LIN {X 0,Y 249.279,Z 155.051,A -85,B 0,C 180,E1 -18895.148,E2 -18895.148} C_VEL
LIN {X 0,Y 249.67,Z 155.011,A -85,B 0,C 180,E1 -18898.387,E2 -18898.387} C_VEL
LIN {X 0,Y 249.663,Z 155.008,A -85,B 0,C 180,E1 -18901.613,E2 -18901.613} C_VEL
LIN {X 0,Y 249.424,Z 155.041,A -85,B 0,C 180,E1 -18906.545,E2 -18906.545} C_VEL
LIN {X 0,Y 249.344,Z 155.042,A -85,B 0,C 180,E1 -18909.737,E2 -18909.737} C_VEL
LIN {X 0,Y 249.16,Z 155.074,A -85,B 0,C 180,E1 -18914.706,E2 -18914.706} C_VEL
LIN {X 0,Y 249.108,Z 155.073,A -85,B 0,C 180,E1 -18918.08,E2 -18918.08} C_VEL
LIN {X 0,Y 249.082,Z 155.075,A -85,B 0,C 180,E1 -18921.519,E2 -18921.519} C_VEL
LIN {X 0,Y 249.086,Z 155.051,A -85,B 0,C 180,E1 -18925.46,E2 -18925.46} C_VEL
LIN {X 0,Y 249.038,Z 155.082,A -85,B 0,C 180,E1 -18928.974,E2 -18928.974} C_VEL
LIN {X 0,Y 249.028,Z 155.089,A -85,B 0,C 180,E1 -18932.426,E2 -18932.426} C_VEL
LIN {X 0,Y 249.046,Z 155.084,A -85,B 0,C 180,E1 -18936.343,E2 -18936.343} C_VEL
LIN {X 0,Y 249.026,Z 155.159,A -85,B 0,C 180,E1 -18939.615,E2 -18939.615} C_VEL
LIN {X 0,Y 249.925,Z 157.806,A -85,B 0,C 180,E1 -18939.982,E2 -18939.982} C_VEL
LIN {X 0,Y 252.085,Z 160.128,A -85,B 0,C 180,E1 -18940.669,E2 -18940.669} C_VEL
LIN {X 0,Y 252.72,Z 160.982,A -85,B 0,C 180,E1 -18940.874,E2 -18940.874} C_VEL
LIN {X 0,Y 254.881,Z 164.177,A -85,B 0,C 180,E1 -18941.57,E2 -18941.57} C_VEL
LIN {X 0,Y 256.285,Z 165.902,A -85,B 0,C 180,E1 -18941.996,E2 -18941.996} C_VEL
LIN {X 0,Y 264.754,Z 177.926,A -85,B 0,C 180,E1 -18944.469,E2 -18944.469} C_VEL
LIN {X 0,Y 273.524,Z 191.575,A -85,B 0,C 180,E1 -18946.809,E2 -18946.809} C_VEL
LIN {X 0,Y 280.062,Z 204.114,A -85,B 0,C 180,E1 -18948.485,E2 -18948.485} C_VEL
LIN {X 0,Y 285.989,Z 217.193,A -85,B 0,C 180,E1 -18949.959,E2 -18949.959} C_VEL
LIN {X 0,Y 281.284,Z 313.77,A -85,B 0,C 180,E1 -18952.312,E2 -18952.312} C_VEL
LIN {X 0,Y 279.771,Z 329.461,A -85,B 0,C 180,E1 -18952.923,E2 -18952.923} C_VEL
LIN {X 0,Y 277.923,Z 343.793,A -85,B 0,C 180,E1 -18953.765,E2 -18953.765} C_VEL
LIN {X 0,Y 275.593,Z 357.91,A -85,B 0,C 180,E1 -18954.874,E2 -18954.874} C_VEL
LIN {X 0,Y 272.986,Z 370.88,A -85,B 0,C 180,E1 -18956.17,E2 -18956.17} C_VEL
LIN {X 0,Y 269.885,Z 383.644,A -85,B 0,C 180,E1 -18957.735,E2 -18957.735} C_VEL
LIN {X 0,Y 266.362,Z 396.502,A -85,B 0,C 180,E1 -18959.694,E2 -18959.694} C_VEL
LIN {X 0,Y 262.829,Z 408.079,A -85,B 0,C 180,E1 -18961.868,E2 -18961.868} C_VEL
LIN {X 0,Y 259.552,Z 418.653,A -85,B 0,C 180,E1 -18964.327,E2 -18964.327} C_VEL
LIN {X 0,Y 256.387,Z 428.094,A -85,B 0,C 180,E1 -18967.007,E2 -18967.007} C_VEL
LIN {X 0,Y 253.645,Z 435.952,A -85,B 0,C 180,E1 -18969.736,E2 -18969.736} C_VEL
LIN {X 0,Y 251.289,Z 443.278,A -85,B 0,C 180,E1 -18972.923,E2 -18972.923} C_VEL
LIN {X 0,Y 249.398,Z 449.09,A -85,B 0,C 180,E1 -18976.141,E2 -18976.141} C_VEL
LIN {X 0,Y 248.473,Z 452.526,A -85,B 0,C 180,E1 -18978.58,E2 -18978.58} C_VEL
LIN {X 0,Y 247.639,Z 456.003,A -85,B 0,C 180,E1 -18981.842,E2 -18981.842} C_VEL
LIN {X 0,Y 247.133,Z 458.3,A -85,B 0,C 180,E1 -18985.106,E2 -18985.106} C_VEL
LIN {X 0,Y 246.994,Z 459.468,A -85,B 0,C 180,E1 -18988.37,E2 -18988.37} C_VEL
LIN {X 0,Y 246.994,Z 459.481,A -85,B 0,C 180,E1 -18991.631,E2 -18991.631} C_VEL
LIN {X 0,Y 247.133,Z 458.365,A -85,B 0,C 180,E1 -18994.894,E2 -18994.894} C_VEL
LIN {X 0,Y 247.628,Z 456.118,A -85,B 0,C 180,E1 -18998.158,E2 -18998.158} C_VEL
LIN {X 0,Y 248.446,Z 452.688,A -85,B 0,C 180,E1 -19001.421,E2 -19001.421} C_VEL
LIN {X 0,Y 249.796,Z 447.987,A -85,B 0,C 180,E1 -19004.668,E2 -19004.668} C_VEL
LIN {X 0,Y 251.742,Z 441.891,A -85,B 0,C 180,E1 -19007.884,E2 -19007.884} C_VEL
LIN {X 0,Y 254.321,Z 434.209,A -85,B 0,C 180,E1 -19011.054,E2 -19011.054} C_VEL
LIN {X 0,Y 257.162,Z 426.014,A -85,B 0,C 180,E1 -19013.773,E2 -19013.773} C_VEL
LIN {X 0,Y 260.532,Z 416.135,A -85,B 0,C 180,E1 -19016.43,E2 -19016.43} C_VEL
LIN {X 0,Y 263.613,Z 406.01,A -85,B 0,C 180,E1 -19018.678,E2 -19018.678} C_VEL
LIN {X 0,Y 266.589,Z 396.072,A -85,B 0,C 180,E1 -19020.496,E2 -19020.496} C_VEL
LIN {X 0,Y 270.04,Z 383.126,A -85,B 0,C 180,E1 -19022.465,E2 -19022.465} C_VEL
LIN {X 0,Y 273.18,Z 370.256,A -85,B 0,C 180,E1 -19024.025,E2 -19024.025} C_VEL
LIN {X 0,Y 275.934,Z 356.158,A -85,B 0,C 180,E1 -19025.409,E2 -19025.409} C_VEL
LIN {X 0,Y 278.343,Z 341.437,A -85,B 0,C 180,E1 -19026.509,E2 -19026.509} C_VEL
LIN {X 0,Y 280.226,Z 326.136,A -85,B 0,C 180,E1 -19027.345,E2 -19027.345} C_VEL
LIN {X 0,Y 281.517,Z 311.329,A -85,B 0,C 180,E1 -19027.878,E2 -19027.878} C_VEL
LIN {X 0,Y 285.259,Z 232.852,A -85,B 0,C 180,E1 -19029.796,E2 -19029.796} C_VEL
LIN {X 0,Y 286.027,Z 216.985,A -85,B 0,C 180,E1 -19030.178,E2 -19030.178} C_VEL
LIN {X 0,Y 278.236,Z 200.326,A -85,B 0,C 180,E1 -19032.122,E2 -19032.122} C_VEL
LIN {X 0,Y 272.973,Z 190.671,A -85,B 0,C 180,E1 -19033.478,E2 -19033.478} C_VEL
LIN {X 0,Y 264.56,Z 177.55,A -85,B 0,C 180,E1 -19035.742,E2 -19035.742} C_VEL
LIN {X 0,Y 258.212,Z 168.659,A -85,B 0,C 180,E1 -19037.575,E2 -19037.575} C_VEL
LIN {X 0,Y 255.212,Z 164.469,A -85,B 0,C 180,E1 -19038.496,E2 -19038.496} C_VEL
LIN {X 0,Y 253.025,Z 161.57,A -85,B 0,C 180,E1 -19039.186,E2 -19039.186} C_VEL
LIN {X 0,Y 252.124,Z 160.16,A -85,B 0,C 180,E1 -19039.486,E2 -19039.486} C_VEL
LIN {X 0,Y 250.043,Z 158.023,A -85,B 0,C 180,E1 -19040.145,E2 -19040.145} C_VEL
LIN {X 0,Y 249.052,Z 155.413,A -85,B 0,C 180,E1 -19040.537,E2 -19040.537} C_VEL
LIN {X 0,Y 248.992,Z 155.088,A -85,B 0,C 180,E1 -19040.574,E2 -19040.574} C_VEL
LIN {X 0,Y 249.044,Z 155.083,A -85,B 0,C 180,E1 -19044.923,E2 -19044.923} C_VEL
LIN {X 0,Y 249.032,Z 155.058,A -85,B 0,C 180,E1 -19047.848,E2 -19047.848} C_VEL
LIN {X 0,Y 249.037,Z 155.083,A -85,B 0,C 180,E1 -19051.331,E2 -19051.331} C_VEL
LIN {X 0,Y 249.058,Z 155.082,A -85,B 0,C 180,E1 -19054.958,E2 -19054.958} C_VEL
LIN {X 0,Y 248.998,Z 155.084,A -85,B 0,C 180,E1 -19057.604,E2 -19057.604} C_VEL
LIN {X 0,Y 248.358,Z 155.171,A -85,B 0,C 180,E1 -19058.954,E2 -19058.954} C_VEL
LIN {X 0,Y 245.535,Z 155.517,A -85,B 0,C 180,E1 -19061.157,E2 -19061.157} C_VEL
LIN {X 0,Y 243.154,Z 155.815,A -85,B 0,C 180,E1 -19062.951,E2 -19062.951} C_VEL
LIN {X 0,Y 242.174,Z 155.944,A -85,B 0,C 180,E1 -19064.342,E2 -19064.342} C_VEL
LIN {X 0,Y 242.118,Z 155.947,A -85,B 0,C 180,E1 -19064.812,E2 -19064.812} C_VEL
LIN {X 0,Y 242.344,Z 155.909,A -85,B 0,C 180,E1 -19070.404,E2 -19070.404} C_VEL
LIN {X 0,Y 242.398,Z 155.917,A -85,B 0,C 180,E1 -19073.34,E2 -19073.34} C_VEL
LIN {X 0,Y 242.622,Z 155.886,A -85,B 0,C 180,E1 -19078.34,E2 -19078.34} C_VEL
LIN {X 0,Y 242.632,Z 155.883,A -85,B 0,C 180,E1 -19081.66,E2 -19081.66} C_VEL
LIN {X 0,Y 242.405,Z 155.915,A -85,B 0,C 180,E1 -19086.659,E2 -19086.659} C_VEL
LIN {X 0,Y 242.269,Z 155.923,A -85,B 0,C 180,E1 -19090.023,E2 -19090.023} C_VEL
LIN {X 0,Y 242.141,Z 155.945,A -85,B 0,C 180,E1 -19095.142,E2 -19095.142} C_VEL
LIN {X 0,Y 242.059,Z 155.949,A -85,B 0,C 180,E1 -19098.625,E2 -19098.625} C_VEL
LIN {X 0,Y 242.006,Z 155.956,A -85,B 0,C 180,E1 -19102.18,E2 -19102.18} C_VEL
LIN {X 0,Y 242.034,Z 155.954,A -85,B 0,C 180,E1 -19105.821,E2 -19105.821} C_VEL
LIN {X 0,Y 241.972,Z 155.969,A -85,B 0,C 180,E1 -19109.588,E2 -19109.588} C_VEL
LIN {X 0,Y 241.98,Z 155.958,A -85,B 0,C 180,E1 -19113.492,E2 -19113.492} C_VEL
LIN {X 0,Y 242.015,Z 156.047,A -85,B 0,C 180,E1 -19115.736,E2 -19115.736} C_VEL
LIN {X 0,Y 243.277,Z 159.716,A -85,B 0,C 180,E1 -19117.625,E2 -19117.625} C_VEL
LIN {X 0,Y 246.451,Z 164.423,A -85,B 0,C 180,E1 -19118.781,E2 -19118.781} C_VEL
LIN {X 0,Y 251.53,Z 172.11,A -85,B 0,C 180,E1 -19120.521,E2 -19120.521} C_VEL
LIN {X 0,Y 257.815,Z 182.158,A -85,B 0,C 180,E1 -19122.525,E2 -19122.525} C_VEL
LIN {X 0,Y 265.356,Z 195.282,A -85,B 0,C 180,E1 -19124.756,E2 -19124.756} C_VEL
LIN {X 0,Y 273.059,Z 210.704,A -85,B 0,C 180,E1 -19126.899,E2 -19126.899} C_VEL
LIN {X 0,Y 279.533,Z 225.506,A -85,B 0,C 180,E1 -19128.619,E2 -19128.619} C_VEL
LIN {X 0,Y 280.218,Z 227.267,A -85,B 0,C 180,E1 -19128.8,E2 -19128.8} C_VEL
LIN {X 0,Y 275.438,Z 323.887,A -85,B 0,C 180,E1 -19131.19,E2 -19131.19} C_VEL
LIN {X 0,Y 273.972,Z 339.511,A -85,B 0,C 180,E1 -19131.767,E2 -19131.767} C_VEL
LIN {X 0,Y 271.831,Z 354.535,A -85,B 0,C 180,E1 -19132.585,E2 -19132.585} C_VEL
LIN {X 0,Y 269.274,Z 368.105,A -85,B 0,C 180,E1 -19133.575,E2 -19133.575} C_VEL
LIN {X 0,Y 266.389,Z 381.613,A -85,B 0,C 180,E1 -19134.871,E2 -19134.871} C_VEL
LIN {X 0,Y 262.91,Z 395.389,A -85,B 0,C 180,E1 -19136.541,E2 -19136.541} C_VEL
LIN {X 0,Y 259.39,Z 407.401,A -85,B 0,C 180,E1 -19138.335,E2 -19138.335} C_VEL
LIN {X 0,Y 255.896,Z 418.533,A -85,B 0,C 180,E1 -19140.372,E2 -19140.372} C_VEL
LIN {X 0,Y 252.486,Z 429.103,A -85,B 0,C 180,E1 -19142.749,E2 -19142.749} C_VEL
LIN {X 0,Y 249.285,Z 438.815,A -85,B 0,C 180,E1 -19145.427,E2 -19145.427} C_VEL
LIN {X 0,Y 246.303,Z 447.143,A -85,B 0,C 180,E1 -19148.226,E2 -19148.226} C_VEL
LIN {X 0,Y 243.715,Z 454.975,A -85,B 0,C 180,E1 -19151.506,E2 -19151.506} C_VEL
LIN {X 0,Y 241.836,Z 461.213,A -85,B 0,C 180,E1 -19154.838,E2 -19154.838} C_VEL
LIN {X 0,Y 240.569,Z 466.043,A -85,B 0,C 180,E1 -19158.2,E2 -19158.2} C_VEL
LIN {X 0,Y 239.938,Z 469.588,A -85,B 0,C 180,E1 -19161.578,E2 -19161.578} C_VEL
LIN {X 0,Y 239.734,Z 472.123,A -85,B 0,C 180,E1 -19165.367,E2 -19165.367} C_VEL
LIN {X 0,Y 239.828,Z 473.101,A -85,B 0,C 180,E1 -19168.321,E2 -19168.321} C_VEL
LIN {X 0,Y 239.89,Z 473.257,A -85,B 0,C 180,E1 -19170,E2 -19170} C_VEL
LIN {X 0,Y 239.743,Z 472.642,A -85,B 0,C 180,E1 -19173.361,E2 -19173.361} C_VEL
LIN {X 0,Y 239.785,Z 470.873,A -85,B 0,C 180,E1 -19176.733,E2 -19176.733} C_VEL
LIN {X 0,Y 240.221,Z 467.929,A -85,B 0,C 180,E1 -19180.11,E2 -19180.11} C_VEL
LIN {X 0,Y 241.154,Z 463.743,A -85,B 0,C 180,E1 -19183.482,E2 -19183.482} C_VEL
LIN {X 0,Y 242.591,Z 458.203,A -85,B 0,C 180,E1 -19186.84,E2 -19186.84} C_VEL
LIN {X 0,Y 244.884,Z 451.171,A -85,B 0,C 180,E1 -19190.145,E2 -19190.145} C_VEL
LIN {X 0,Y 247.87,Z 442.43,A -85,B 0,C 180,E1 -19193.388,E2 -19193.388} C_VEL
LIN {X 0,Y 250.802,Z 433.768,A -85,B 0,C 180,E1 -19196.004,E2 -19196.004} C_VEL
LIN {X 0,Y 254.136,Z 423.717,A -85,B 0,C 180,E1 -19198.492,E2 -19198.492} C_VEL
LIN {X 0,Y 258.072,Z 411.491,A -85,B 0,C 180,E1 -19200.932,E2 -19200.932} C_VEL
LIN {X 0,Y 261.822,Z 399.029,A -85,B 0,C 180,E1 -19202.927,E2 -19202.927} C_VEL
LIN {X 0,Y 265.257,Z 386.188,A -85,B 0,C 180,E1 -19204.586,E2 -19204.586} C_VEL
LIN {X 0,Y 268.498,Z 371.686,A -85,B 0,C 180,E1 -19206.082,E2 -19206.082} C_VEL
LIN {X 0,Y 271.35,Z 356.628,A -85,B 0,C 180,E1 -19207.259,E2 -19207.259} C_VEL
LIN {X 0,Y 273.622,Z 341.541,A -85,B 0,C 180,E1 -19208.115,E2 -19208.115} C_VEL
LIN {X 0,Y 275.223,Z 325.688,A -85,B 0,C 180,E1 -19208.728,E2 -19208.728} C_VEL
LIN {X 0,Y 280.137,Z 228.134,A -85,B 0,C 180,E1 -19211.137,E2 -19211.137} C_VEL
LIN {X 0,Y 279.833,Z 226.451,A -85,B 0,C 180,E1 -19211.247,E2 -19211.247} C_VEL
LIN {X 0,Y 273.593,Z 211.928,A -85,B 0,C 180,E1 -19212.9,E2 -19212.9} C_VEL
LIN {X 0,Y 266.604,Z 197.759,A -85,B 0,C 180,E1 -19214.824,E2 -19214.824} C_VEL
LIN {X 0,Y 259.313,Z 184.701,A -85,B 0,C 180,E1 -19216.95,E2 -19216.95} C_VEL
LIN {X 0,Y 253.146,Z 174.691,A -85,B 0,C 180,E1 -19218.873,E2 -19218.873} C_VEL
LIN {X 0,Y 249.875,Z 169.56,A -85,B 0,C 180,E1 -19219.956,E2 -19219.956} C_VEL
LIN {X 0,Y 246.144,Z 164.055,A -85,B 0,C 180,E1 -19221.242,E2 -19221.242} C_VEL
LIN {X 0,Y 243.202,Z 159.541,A -85,B 0,C 180,E1 -19222.319,E2 -19222.319} C_VEL
LIN {X 0,Y 242.005,Z 155.955,A -85,B 0,C 180,E1 -19224.263,E2 -19224.263} C_VEL
LIN {X 0,Y 241.977,Z 155.966,A -85,B 0,C 180,E1 -19228.48,E2 -19228.48} C_VEL
LIN {X 0,Y 242.01,Z 155.959,A -85,B 0,C 180,E1 -19232.313,E2 -19232.313} C_VEL
LIN {X 0,Y 242.059,Z 155.951,A -85,B 0,C 180,E1 -19236.016,E2 -19236.016} C_VEL
LIN {X 0,Y 242.039,Z 155.952,A -85,B 0,C 180,E1 -19239.608,E2 -19239.608} C_VEL
LIN {X 0,Y 242.165,Z 155.936,A -85,B 0,C 180,E1 -19243.278,E2 -19243.278} C_VEL
LIN {X 0,Y 242.152,Z 155.94,A -85,B 0,C 180,E1 -19246.574,E2 -19246.574} C_VEL
LIN {X 0,Y 242.343,Z 155.919,A -85,B 0,C 180,E1 -19250.405,E2 -19250.405} C_VEL
LIN {X 0,Y 242.4,Z 155.916,A -85,B 0,C 180,E1 -19253.34,E2 -19253.34} C_VEL
LIN {X 0,Y 242.631,Z 155.888,A -85,B 0,C 180,E1 -19258.34,E2 -19258.34} C_VEL
LIN {X 0,Y 242.623,Z 155.885,A -85,B 0,C 180,E1 -19261.66,E2 -19261.66} C_VEL
LIN {X 0,Y 242.399,Z 155.917,A -85,B 0,C 180,E1 -19266.66,E2 -19266.66} C_VEL
LIN {X 0,Y 242.267,Z 155.926,A -85,B 0,C 180,E1 -19270.024,E2 -19270.024} C_VEL
LIN {X 0,Y 242.114,Z 155.952,A -85,B 0,C 180,E1 -19275.144,E2 -19275.144} C_VEL
LIN {X 0,Y 242.047,Z 155.958,A -85,B 0,C 180,E1 -19278.626,E2 -19278.626} C_VEL
LIN {X 0,Y 242.005,Z 155.961,A -85,B 0,C 180,E1 -19282.181,E2 -19282.181} C_VEL
LIN {X 0,Y 242.034,Z 155.926,A -85,B 0,C 180,E1 -19285.821,E2 -19285.821} C_VEL
LIN {X 0,Y 241.97,Z 155.97,A -85,B 0,C 180,E1 -19289.588,E2 -19289.588} C_VEL
LIN {X 0,Y 241.98,Z 155.964,A -85,B 0,C 180,E1 -19293.493,E2 -19293.493} C_VEL
LIN {X 0,Y 241.995,Z 155.966,A -85,B 0,C 180,E1 -19297.581,E2 -19297.581} C_VEL
LIN {X 0,Y 242.867,Z 158.603,A -85,B 0,C 180,E1 -19297.974,E2 -19297.974} C_VEL
LIN {X 0,Y 244.856,Z 160.844,A -85,B 0,C 180,E1 -19298.675,E2 -19298.675} C_VEL
LIN {X 0,Y 245.688,Z 161.619,A -85,B 0,C 180,E1 -19298.954,E2 -19298.954} C_VEL
LIN {X 0,Y 247.867,Z 165.014,A -85,B 0,C 180,E1 -19299.73,E2 -19299.73} C_VEL
LIN {X 0,Y 249.467,Z 166.854,A -85,B 0,C 180,E1 -19300.254,E2 -19300.254} C_VEL
LIN {X 0,Y 252.09,Z 170.381,A -85,B 0,C 180,E1 -19301.109,E2 -19301.109} C_VEL
LIN {X 0,Y 261.02,Z 183.198,A -85,B 0,C 180,E1 -19303.827,E2 -19303.827} C_VEL
LIN {X 0,Y 269.645,Z 196.844,A -85,B 0,C 180,E1 -19306.216,E2 -19306.216} C_VEL
LIN {X 0,Y 276.191,Z 209.815,A -85,B 0,C 180,E1 -19307.961,E2 -19307.961} C_VEL
LIN {X 0,Y 280.5,Z 219.373,A -85,B 0,C 180,E1 -19309.075,E2 -19309.075} C_VEL
LIN {X 0,Y 275.708,Z 313.988,A -85,B 0,C 180,E1 -19311.411,E2 -19311.411} C_VEL
LIN {X 0,Y 274.139,Z 329.672,A -85,B 0,C 180,E1 -19312.028,E2 -19312.028} C_VEL
LIN {X 0,Y 272.063,Z 345.291,A -85,B 0,C 180,E1 -19312.971,E2 -19312.971} C_VEL
LIN {X 0,Y 269.525,Z 359.809,A -85,B 0,C 180,E1 -19314.159,E2 -19314.159} C_VEL
LIN {X 0,Y 266.398,Z 374.215,A -85,B 0,C 180,E1 -19315.674,E2 -19315.674} C_VEL
LIN {X 0,Y 262.879,Z 387.666,A -85,B 0,C 180,E1 -19317.45,E2 -19317.45} C_VEL
LIN {X 0,Y 259.283,Z 399.872,A -85,B 0,C 180,E1 -19319.454,E2 -19319.454} C_VEL
LIN {X 0,Y 255.626,Z 411.397,A -85,B 0,C 180,E1 -19321.798,E2 -19321.798} C_VEL
LIN {X 0,Y 252.133,Z 421.778,A -85,B 0,C 180,E1 -19324.402,E2 -19324.402} C_VEL
LIN {X 0,Y 249.01,Z 430.732,A -85,B 0,C 180,E1 -19327.165,E2 -19327.165} C_VEL
LIN {X 0,Y 246.233,Z 438.153,A -85,B 0,C 180,E1 -19329.97,E2 -19329.97} C_VEL
LIN {X 0,Y 243.968,Z 445.077,A -85,B 0,C 180,E1 -19333.258,E2 -19333.258} C_VEL
LIN {X 0,Y 242.116,Z 450.518,A -85,B 0,C 180,E1 -19336.572,E2 -19336.572} C_VEL
LIN {X 0,Y 240.984,Z 454.617,A -85,B 0,C 180,E1 -19339.922,E2 -19339.922} C_VEL
LIN {X 0,Y 240.273,Z 457.494,A -85,B 0,C 180,E1 -19343.281,E2 -19343.281} C_VEL
LIN {X 0,Y 239.977,Z 459.221,A -85,B 0,C 180,E1 -19346.642,E2 -19346.642} C_VEL
LIN {X 0,Y 239.922,Z 459.821,A -85,B 0,C 180,E1 -19350,E2 -19350} C_VEL
LIN {X 0,Y 239.977,Z 459.259,A -85,B 0,C 180,E1 -19353.358,E2 -19353.358} C_VEL
LIN {X 0,Y 240.273,Z 457.584,A -85,B 0,C 180,E1 -19356.719,E2 -19356.719} C_VEL
LIN {X 0,Y 240.943,Z 454.755,A -85,B 0,C 180,E1 -19360.079,E2 -19360.079} C_VEL
LIN {X 0,Y 242.07,Z 450.702,A -85,B 0,C 180,E1 -19363.43,E2 -19363.43} C_VEL
LIN {X 0,Y 243.928,Z 445.319,A -85,B 0,C 180,E1 -19366.745,E2 -19366.745} C_VEL
LIN {X 0,Y 246.216,Z 438.462,A -85,B 0,C 180,E1 -19370.031,E2 -19370.031} C_VEL
LIN {X 0,Y 249.294,Z 429.892,A -85,B 0,C 180,E1 -19373.246,E2 -19373.246} C_VEL
LIN {X 0,Y 252.548,Z 420.775,A -85,B 0,C 180,E1 -19375.995,E2 -19375.995} C_VEL
LIN {X 0,Y 255.556,Z 411.941,A -85,B 0,C 180,E1 -19378.194,E2 -19378.194} C_VEL
LIN {X 0,Y 259.144,Z 400.45,A -85,B 0,C 180,E1 -19380.564,E2 -19380.564} C_VEL
LIN {X 0,Y 262.729,Z 388.354,A -85,B 0,C 180,E1 -19382.571,E2 -19382.571} C_VEL
LIN {X 0,Y 265.927,Z 376.485,A -85,B 0,C 180,E1 -19384.167,E2 -19384.167} C_VEL
LIN {X 0,Y 268.756,Z 363.809,A -85,B 0,C 180,E1 -19385.578,E2 -19385.578} C_VEL
LIN {X 0,Y 271.362,Z 350.032,A -85,B 0,C 180,E1 -19386.792,E2 -19386.792} C_VEL
LIN {X 0,Y 273.568,Z 335.39,A -85,B 0,C 180,E1 -19387.774,E2 -19387.774} C_VEL
LIN {X 0,Y 275.265,Z 320.346,A -85,B 0,C 180,E1 -19388.487,E2 -19388.487} C_VEL
LIN {X 0,Y 276.424,Z 303.318,A -85,B 0,C 180,E1 -19388.996,E2 -19388.996} C_VEL
LIN {X 0,Y 280.525,Z 219.259,A -85,B 0,C 180,E1 -19391.063,E2 -19391.063} C_VEL
LIN {X 0,Y 272.917,Z 202.924,A -85,B 0,C 180,E1 -19393.054,E2 -19393.054} C_VEL
LIN {X 0,Y 267.7,Z 193.547,A -85,B 0,C 180,E1 -19394.458,E2 -19394.458} C_VEL
LIN {X 0,Y 259.333,Z 180.741,A -85,B 0,C 180,E1 -19396.82,E2 -19396.82} C_VEL
LIN {X 0,Y 254.1,Z 173.341,A -85,B 0,C 180,E1 -19398.409,E2 -19398.409} C_VEL
LIN {X 0,Y 251.807,Z 170.056,A -85,B 0,C 180,E1 -19399.145,E2 -19399.145} C_VEL
LIN {X 0,Y 249.225,Z 166.389,A -85,B 0,C 180,E1 -19400.002,E2 -19400.002} C_VEL
LIN {X 0,Y 246.478,Z 163.164,A -85,B 0,C 180,E1 -19400.92,E2 -19400.92} C_VEL
LIN {X 0,Y 245.414,Z 161.207,A -85,B 0,C 180,E1 -19401.319,E2 -19401.319} C_VEL
LIN {X 0,Y 243.17,Z 159.063,A -85,B 0,C 180,E1 -19402.09,E2 -19402.09} C_VEL
LIN {X 0,Y 242.146,Z 156.808,A -85,B 0,C 180,E1 -19402.512,E2 -19402.512} C_VEL
LIN {X 0,Y 241.958,Z 155.942,A -85,B 0,C 180,E1 -19402.642,E2 -19402.642} C_VEL
LIN {X 0,Y 241.98,Z 155.955,A -85,B 0,C 180,E1 -19406.507,E2 -19406.507} C_VEL
LIN {X 0,Y 241.972,Z 155.948,A -85,B 0,C 180,E1 -19410.615,E2 -19410.615} C_VEL
LIN {X 0,Y 241.997,Z 155.957,A -85,B 0,C 180,E1 -19414.197,E2 -19414.197} C_VEL
LIN {X 0,Y 241.987,Z 155.958,A -85,B 0,C 180,E1 -19418.338,E2 -19418.338} C_VEL
LIN {X 0,Y 242.115,Z 155.949,A -85,B 0,C 180,E1 -19423.318,E2 -19423.318} C_VEL
LIN {X 0,Y 242.118,Z 155.947,A -85,B 0,C 180,E1 -19424.812,E2 -19424.812} C_VEL
LIN {X 0,Y 241.526,Z 156.027,A -85,B 0,C 180,E1 -19426.202,E2 -19426.202} C_VEL
LIN {X 0,Y 238.758,Z 156.37,A -85,B 0,C 180,E1 -19428.472,E2 -19428.472} C_VEL
LIN {X 0,Y 236.381,Z 156.655,A -85,B 0,C 180,E1 -19430.321,E2 -19430.321} C_VEL
LIN {X 0,Y 235.376,Z 156.781,A -85,B 0,C 180,E1 -19431.754,E2 -19431.754} C_VEL
LIN {X 0,Y 235.304,Z 156.79,A -85,B 0,C 180,E1 -19432.24,E2 -19432.24} C_VEL
LIN {X 0,Y 235.581,Z 156.764,A -85,B 0,C 180,E1 -19438.29,E2 -19438.29} C_VEL
LIN {X 0,Y 235.591,Z 156.76,A -85,B 0,C 180,E1 -19441.709,E2 -19441.709} C_VEL
LIN {X 0,Y 235.357,Z 156.794,A -85,B 0,C 180,E1 -19446.86,E2 -19446.86} C_VEL
LIN {X 0,Y 235.216,Z 156.803,A -85,B 0,C 180,E1 -19450.327,E2 -19450.327} C_VEL
LIN {X 0,Y 235.088,Z 156.829,A -85,B 0,C 180,E1 -19455.608,E2 -19455.608} C_VEL
LIN {X 0,Y 234.999,Z 156.832,A -85,B 0,C 180,E1 -19459.206,E2 -19459.206} C_VEL
LIN {X 0,Y 234.951,Z 156.835,A -85,B 0,C 180,E1 -19462.884,E2 -19462.884} C_VEL
LIN {X 0,Y 234.948,Z 156.834,A -85,B 0,C 180,E1 -19466.66,E2 -19466.66} C_VEL
LIN {X 0,Y 234.901,Z 156.85,A -85,B 0,C 180,E1 -19470.572,E2 -19470.572} C_VEL
LIN {X 0,Y 234.953,Z 156.98,A -85,B 0,C 180,E1 -19473.896,E2 -19473.896} C_VEL
LIN {X 0,Y 235.708,Z 159.293,A -85,B 0,C 180,E1 -19475.163,E2 -19475.163} C_VEL
LIN {X 0,Y 239.209,Z 164.253,A -85,B 0,C 180,E1 -19476.574,E2 -19476.574} C_VEL
LIN {X 0,Y 244.827,Z 172.493,A -85,B 0,C 180,E1 -19478.679,E2 -19478.679} C_VEL
LIN {X 0,Y 248.268,Z 177.891,A -85,B 0,C 180,E1 -19479.893,E2 -19479.893} C_VEL
LIN {X 0,Y 254.035,Z 187.247,A -85,B 0,C 180,E1 -19481.804,E2 -19481.804} C_VEL
LIN {X 0,Y 261.151,Z 199.822,A -85,B 0,C 180,E1 -19484,E2 -19484} C_VEL
LIN {X 0,Y 268.925,Z 215.645,A -85,B 0,C 180,E1 -19486.253,E2 -19486.253} C_VEL
LIN {X 0,Y 274.781,Z 229.379,A -85,B 0,C 180,E1 -19487.878,E2 -19487.878} C_VEL
LIN {X 0,Y 270.599,Z 311.991,A -85,B 0,C 180,E1 -19489.937,E2 -19489.937} C_VEL
LIN {X 0,Y 269.322,Z 331.334,A -85,B 0,C 180,E1 -19490.5,E2 -19490.5} C_VEL
LIN {X 0,Y 267.41,Z 346.7,A -85,B 0,C 180,E1 -19491.196,E2 -19491.196} C_VEL
LIN {X 0,Y 264.858,Z 361.541,A -85,B 0,C 180,E1 -19492.148,E2 -19492.148} C_VEL
LIN {X 0,Y 261.969,Z 375.458,A -85,B 0,C 180,E1 -19493.351,E2 -19493.351} C_VEL
LIN {X 0,Y 258.562,Z 389.504,A -85,B 0,C 180,E1 -19494.92,E2 -19494.92} C_VEL
LIN {X 0,Y 254.73,Z 402.636,A -85,B 0,C 180,E1 -19496.746,E2 -19496.746} C_VEL
LIN {X 0,Y 250.993,Z 414.47,A -85,B 0,C 180,E1 -19498.801,E2 -19498.801} C_VEL
LIN {X 0,Y 247.311,Z 425.318,A -85,B 0,C 180,E1 -19501.112,E2 -19501.112} C_VEL
LIN {X 0,Y 243.652,Z 436.004,A -85,B 0,C 180,E1 -19503.941,E2 -19503.941} C_VEL
LIN {X 0,Y 240.458,Z 444.694,A -85,B 0,C 180,E1 -19506.76,E2 -19506.76} C_VEL
LIN {X 0,Y 238.16,Z 451.072,A -85,B 0,C 180,E1 -19509.261,E2 -19509.261} C_VEL
LIN {X 0,Y 235.824,Z 458.08,A -85,B 0,C 180,E1 -19512.661,E2 -19512.661} C_VEL
LIN {X 0,Y 234.202,Z 463.596,A -85,B 0,C 180,E1 -19516.109,E2 -19516.109} C_VEL
LIN {X 0,Y 233.167,Z 467.771,A -85,B 0,C 180,E1 -19519.581,E2 -19519.581} C_VEL
LIN {X 0,Y 232.705,Z 470.704,A -85,B 0,C 180,E1 -19523.061,E2 -19523.061} C_VEL
LIN {X 0,Y 232.651,Z 472.456,A -85,B 0,C 180,E1 -19526.536,E2 -19526.536} C_VEL
LIN {X 0,Y 232.801,Z 473.058,A -85,B 0,C 180,E1 -19530,E2 -19530} C_VEL
LIN {X 0,Y 232.651,Z 472.443,A -85,B 0,C 180,E1 -19533.464,E2 -19533.464} C_VEL
LIN {X 0,Y 232.705,Z 470.673,A -85,B 0,C 180,E1 -19536.939,E2 -19536.939} C_VEL
LIN {X 0,Y 233.166,Z 467.727,A -85,B 0,C 180,E1 -19540.419,E2 -19540.419} C_VEL
LIN {X 0,Y 234.189,Z 463.541,A -85,B 0,C 180,E1 -19543.891,E2 -19543.891} C_VEL
LIN {X 0,Y 235.804,Z 457.717,A -85,B 0,C 180,E1 -19547.496,E2 -19547.496} C_VEL
LIN {X 0,Y 238.155,Z 450.969,A -85,B 0,C 180,E1 -19550.74,E2 -19550.74} C_VEL
LIN {X 0,Y 240.836,Z 443.452,A -85,B 0,C 180,E1 -19553.656,E2 -19553.656} C_VEL
LIN {X 0,Y 243.906,Z 434.883,A -85,B 0,C 180,E1 -19556.362,E2 -19556.362} C_VEL
LIN {X 0,Y 247.304,Z 425.156,A -85,B 0,C 180,E1 -19558.889,E2 -19558.889} C_VEL
LIN {X 0,Y 250.965,Z 414.277,A -85,B 0,C 180,E1 -19561.203,E2 -19561.203} C_VEL
LIN {X 0,Y 254.725,Z 402.408,A -85,B 0,C 180,E1 -19563.255,E2 -19563.255} C_VEL
LIN {X 0,Y 258.549,Z 389.316,A -85,B 0,C 180,E1 -19565.065,E2 -19565.065} C_VEL
LIN {X 0,Y 261.569,Z 376.858,A -85,B 0,C 180,E1 -19566.475,E2 -19566.475} C_VEL
LIN {X 0,Y 264.43,Z 363.34,A -85,B 0,C 180,E1 -19567.683,E2 -19567.683} C_VEL
LIN {X 0,Y 267.076,Z 348.377,A -85,B 0,C 180,E1 -19568.68,E2 -19568.68} C_VEL
LIN {X 0,Y 268.965,Z 333.822,A -85,B 0,C 180,E1 -19569.38,E2 -19569.38} C_VEL
LIN {X 0,Y 270.196,Z 317.66,A -85,B 0,C 180,E1 -19569.891,E2 -19569.891} C_VEL
LIN {X 0,Y 274.664,Z 229.275,A -85,B 0,C 180,E1 -19572.095,E2 -19572.095} C_VEL
LIN {X 0,Y 268.778,Z 215.5,A -85,B 0,C 180,E1 -19573.725,E2 -19573.725} C_VEL
LIN {X 0,Y 262.197,Z 201.997,A -85,B 0,C 180,E1 -19575.619,E2 -19575.619} C_VEL
LIN {X 0,Y 255.557,Z 189.85,A -85,B 0,C 180,E1 -19577.642,E2 -19577.642} C_VEL
LIN {X 0,Y 249.108,Z 179.249,A -85,B 0,C 180,E1 -19579.741,E2 -19579.741} C_VEL
LIN {X 0,Y 246.409,Z 174.935,A -85,B 0,C 180,E1 -19580.675,E2 -19580.675} C_VEL
LIN {X 0,Y 242.638,Z 169.284,A -85,B 0,C 180,E1 -19582.031,E2 -19582.031} C_VEL
LIN {X 0,Y 239.165,Z 164.145,A -85,B 0,C 180,E1 -19583.352,E2 -19583.352} C_VEL
LIN {X 0,Y 235.967,Z 159.707,A -85,B 0,C 180,E1 -19584.628,E2 -19584.628} C_VEL
LIN {X 0,Y 235.483,Z 158.828,A -85,B 0,C 180,E1 -19584.936,E2 -19584.936} C_VEL
LIN {X 0,Y 234.93,Z 156.839,A -85,B 0,C 180,E1 -19586.203,E2 -19586.203} C_VEL
LIN {X 0,Y 234.971,Z 156.831,A -85,B 0,C 180,E1 -19590.157,E2 -19590.157} C_VEL
LIN {X 0,Y 234.995,Z 156.831,A -85,B 0,C 180,E1 -19593.794,E2 -19593.794} C_VEL
LIN {X 0,Y 235.013,Z 156.831,A -85,B 0,C 180,E1 -19598.97,E2 -19598.97} C_VEL
LIN {X 0,Y 235.098,Z 156.817,A -85,B 0,C 180,E1 -19603.06,E2 -19603.06} C_VEL
LIN {X 0,Y 235.106,Z 156.814,A -85,B 0,C 180,E1 -19607.922,E2 -19607.922} C_VEL
LIN {X 0,Y 235.313,Z 156.787,A -85,B 0,C 180,E1 -19611.412,E2 -19611.412} C_VEL
LIN {X 0,Y 235.351,Z 156.791,A -85,B 0,C 180,E1 -19613.14,E2 -19613.14} C_VEL
LIN {X 0,Y 235.591,Z 156.765,A -85,B 0,C 180,E1 -19618.291,E2 -19618.291} C_VEL
LIN {X 0,Y 235.581,Z 156.763,A -85,B 0,C 180,E1 -19621.71,E2 -19621.71} C_VEL
LIN {X 0,Y 235.35,Z 156.794,A -85,B 0,C 180,E1 -19626.86,E2 -19626.86} C_VEL
LIN {X 0,Y 235.213,Z 156.807,A -85,B 0,C 180,E1 -19630.328,E2 -19630.328} C_VEL
LIN {X 0,Y 235.066,Z 156.829,A -85,B 0,C 180,E1 -19635.61,E2 -19635.61} C_VEL
LIN {X 0,Y 234.989,Z 156.84,A -85,B 0,C 180,E1 -19639.207,E2 -19639.207} C_VEL
LIN {X 0,Y 234.947,Z 156.845,A -85,B 0,C 180,E1 -19642.884,E2 -19642.884} C_VEL
LIN {X 0,Y 234.946,Z 156.807,A -85,B 0,C 180,E1 -19646.66,E2 -19646.66} C_VEL
LIN {X 0,Y 234.9,Z 156.846,A -85,B 0,C 180,E1 -19650.573,E2 -19650.573} C_VEL
LIN {X 0,Y 234.93,Z 156.838,A -85,B 0,C 180,E1 -19654.638,E2 -19654.638} C_VEL
LIN {X 0,Y 234.941,Z 156.864,A -85,B 0,C 180,E1 -19655.313,E2 -19655.313} C_VEL
LIN {X 0,Y 235.76,Z 159.341,A -85,B 0,C 180,E1 -19655.722,E2 -19655.722} C_VEL
LIN {X 0,Y 237.753,Z 161.641,A -85,B 0,C 180,E1 -19656.505,E2 -19656.505} C_VEL
LIN {X 0,Y 238.842,Z 162.527,A -85,B 0,C 180,E1 -19656.903,E2 -19656.903} C_VEL
LIN {X 0,Y 240.78,Z 165.718,A -85,B 0,C 180,E1 -19657.672,E2 -19657.672} C_VEL
LIN {X 0,Y 242.623,Z 167.696,A -85,B 0,C 180,E1 -19658.329,E2 -19658.329} C_VEL
LIN {X 0,Y 245.298,Z 171.406,A -85,B 0,C 180,E1 -19659.288,E2 -19659.288} C_VEL
LIN {X 0,Y 252.299,Z 181.076,A -85,B 0,C 180,E1 -19661.617,E2 -19661.617} C_VEL
LIN {X 0,Y 260.424,Z 193.374,A -85,B 0,C 180,E1 -19664.087,E2 -19664.087} C_VEL
LIN {X 0,Y 266.474,Z 203.452,A -85,B 0,C 180,E1 -19665.798,E2 -19665.798} C_VEL
LIN {X 0,Y 273.417,Z 217.936,A -85,B 0,C 180,E1 -19667.715,E2 -19667.715} C_VEL
LIN {X 0,Y 275.057,Z 221.604,A -85,B 0,C 180,E1 -19668.154,E2 -19668.154} C_VEL
LIN {X 0,Y 270.201,Z 314.207,A -85,B 0,C 180,E1 -19670.473,E2 -19670.473} C_VEL
LIN {X 0,Y 268.578,Z 329.883,A -85,B 0,C 180,E1 -19671.096,E2 -19671.096} C_VEL
LIN {X 0,Y 266.435,Z 345.498,A -85,B 0,C 180,E1 -19672.053,E2 -19672.053} C_VEL
LIN {X 0,Y 264.044,Z 358.614,A -85,B 0,C 180,E1 -19673.126,E2 -19673.126} C_VEL
LIN {X 0,Y 260.945,Z 372.866,A -85,B 0,C 180,E1 -19674.616,E2 -19674.616} C_VEL
LIN {X 0,Y 257.284,Z 386.624,A -85,B 0,C 180,E1 -19676.416,E2 -19676.416} C_VEL
LIN {X 0,Y 253.521,Z 399.036,A -85,B 0,C 180,E1 -19678.45,E2 -19678.45} C_VEL
LIN {X 0,Y 249.703,Z 410.423,A -85,B 0,C 180,E1 -19680.752,E2 -19680.752} C_VEL
LIN {X 0,Y 246.826,Z 419.055,A -85,B 0,C 180,E1 -19682.898,E2 -19682.898} C_VEL
LIN {X 0,Y 243.328,Z 428.497,A -85,B 0,C 180,E1 -19685.696,E2 -19685.696} C_VEL
LIN {X 0,Y 240.334,Z 436.354,A -85,B 0,C 180,E1 -19688.56,E2 -19688.56} C_VEL
LIN {X 0,Y 238.224,Z 442.015,A -85,B 0,C 180,E1 -19691.064,E2 -19691.064} C_VEL
LIN {X 0,Y 236.085,Z 448.174,A -85,B 0,C 180,E1 -19694.459,E2 -19694.459} C_VEL
LIN {X 0,Y 234.527,Z 452.927,A -85,B 0,C 180,E1 -19697.891,E2 -19697.891} C_VEL
LIN {X 0,Y 233.558,Z 456.402,A -85,B 0,C 180,E1 -19701.347,E2 -19701.347} C_VEL
LIN {X 0,Y 232.989,Z 458.698,A -85,B 0,C 180,E1 -19704.808,E2 -19704.808} C_VEL
LIN {X 0,Y 232.821,Z 459.865,A -85,B 0,C 180,E1 -19708.27,E2 -19708.27} C_VEL
LIN {X 0,Y 232.821,Z 459.878,A -85,B 0,C 180,E1 -19711.73,E2 -19711.73} C_VEL
LIN {X 0,Y 233.03,Z 458.585,A -85,B 0,C 180,E1 -19715.581,E2 -19715.581} C_VEL
LIN {X 0,Y 233.526,Z 456.516,A -85,B 0,C 180,E1 -19718.655,E2 -19718.655} C_VEL
LIN {X 0,Y 234.471,Z 453.086,A -85,B 0,C 180,E1 -19722.112,E2 -19722.112} C_VEL
LIN {X 0,Y 236.058,Z 448.383,A -85,B 0,C 180,E1 -19725.543,E2 -19725.543} C_VEL
LIN {X 0,Y 238.185,Z 442.288,A -85,B 0,C 180,E1 -19728.94,E2 -19728.94} C_VEL
LIN {X 0,Y 241.054,Z 434.605,A -85,B 0,C 180,E1 -19732.273,E2 -19732.273} C_VEL
LIN {X 0,Y 244.171,Z 426.409,A -85,B 0,C 180,E1 -19735.122,E2 -19735.122} C_VEL
LIN {X 0,Y 247.856,Z 416.528,A -85,B 0,C 180,E1 -19737.896,E2 -19737.896} C_VEL
LIN {X 0,Y 251.188,Z 406.404,A -85,B 0,C 180,E1 -19740.24,E2 -19740.24} C_VEL
LIN {X 0,Y 254.768,Z 395.398,A -85,B 0,C 180,E1 -19742.309,E2 -19742.309} C_VEL
LIN {X 0,Y 258.176,Z 383.515,A -85,B 0,C 180,E1 -19744.156,E2 -19744.156} C_VEL
LIN {X 0,Y 261.528,Z 370.643,A -85,B 0,C 180,E1 -19745.767,E2 -19745.767} C_VEL
LIN {X 0,Y 264.531,Z 356.387,A -85,B 0,C 180,E1 -19747.203,E2 -19747.203} C_VEL
LIN {X 0,Y 267.062,Z 341.817,A -85,B 0,C 180,E1 -19748.322,E2 -19748.322} C_VEL
LIN {X 0,Y 269.105,Z 326.508,A -85,B 0,C 180,E1 -19749.175,E2 -19749.175} C_VEL
LIN {X 0,Y 270.458,Z 311.686,A -85,B 0,C 180,E1 -19749.724,E2 -19749.724} C_VEL
LIN {X 0,Y 274.52,Z 233.122,A -85,B 0,C 180,E1 -19751.693,E2 -19751.693} C_VEL
LIN {X 0,Y 275.093,Z 221.513,A -85,B 0,C 180,E1 -19751.985,E2 -19751.985} C_VEL
LIN {X 0,Y 267.918,Z 206.173,A -85,B 0,C 180,E1 -19753.949,E2 -19753.949} C_VEL
LIN {X 0,Y 263.328,Z 197.924,A -85,B 0,C 180,E1 -19755.238,E2 -19755.238} C_VEL
LIN {X 0,Y 254.473,Z 184.151,A -85,B 0,C 180,E1 -19757.865,E2 -19757.865} C_VEL
LIN {X 0,Y 248.007,Z 175.1,A -85,B 0,C 180,E1 -19759.953,E2 -19759.953} C_VEL
LIN {X 0,Y 245.099,Z 171.196,A -85,B 0,C 180,E1 -19760.952,E2 -19760.952} C_VEL
LIN {X 0,Y 242.514,Z 167.487,A -85,B 0,C 180,E1 -19761.891,E2 -19761.891} C_VEL
LIN {X 0,Y 239.586,Z 164.024,A -85,B 0,C 180,E1 -19762.968,E2 -19762.968} C_VEL
LIN {X 0,Y 238.588,Z 162.178,A -85,B 0,C 180,E1 -19763.38,E2 -19763.38} C_VEL
LIN {X 0,Y 236.265,Z 160.169,A -85,B 0,C 180,E1 -19764.253,E2 -19764.253} C_VEL
LIN {X 0,Y 235.06,Z 157.602,A -85,B 0,C 180,E1 -19764.799,E2 -19764.799} C_VEL
LIN {X 0,Y 234.929,Z 156.839,A -85,B 0,C 180,E1 -19764.944,E2 -19764.944} C_VEL
LIN {X 0,Y 234.953,Z 156.814,A -85,B 0,C 180,E1 -19767.423,E2 -19767.423} C_VEL
LIN {X 0,Y 234.893,Z 156.844,A -85,B 0,C 180,E1 -19771.398,E2 -19771.398} C_VEL
LIN {X 0,Y 234.916,Z 156.845,A -85,B 0,C 180,E1 -19775.238,E2 -19775.238} C_VEL
LIN {X 0,Y 234.938,Z 156.84,A -85,B 0,C 180,E1 -19778.963,E2 -19778.963} C_VEL
LIN {X 0,Y 235.057,Z 156.825,A -85,B 0,C 180,E1 -19783.093,E2 -19783.093} C_VEL
LIN {X 0,Y 235.1,Z 156.823,A -85,B 0,C 180,E1 -19787.921,E2 -19787.921} C_VEL
LIN {X 0,Y 235.313,Z 156.786,A -85,B 0,C 180,E1 -19791.412,E2 -19791.412} C_VEL
LIN {X 0,Y 235.304,Z 156.79,A -85,B 0,C 180,E1 -19792.24,E2 -19792.24} C_VEL
LIN {X 0,Y 234.672,Z 156.878,A -85,B 0,C 180,E1 -19793.667,E2 -19793.667} C_VEL
LIN {X 0,Y 231.891,Z 157.222,A -85,B 0,C 180,E1 -19795.999,E2 -19795.999} C_VEL
LIN {X 0,Y 229.557,Z 157.516,A -85,B 0,C 180,E1 -19797.9,E2 -19797.9} C_VEL
LIN {X 0,Y 228.614,Z 157.621,A -85,B 0,C 180,E1 -19799.373,E2 -19799.373} C_VEL
LIN {X 0,Y 228.569,Z 157.624,A -85,B 0,C 180,E1 -19799.872,E2 -19799.872} C_VEL
LIN {X 0,Y 228.55,Z 157.638,A -85,B 0,C 180,E1 -19801.762,E2 -19801.762} C_VEL
LIN {X 0,Y 228.309,Z 157.673,A -85,B 0,C 180,E1 -19807.073,E2 -19807.073} C_VEL
LIN {X 0,Y 228.147,Z 157.687,A -85,B 0,C 180,E1 -19810.651,E2 -19810.651} C_VEL
LIN {X 0,Y 228.05,Z 157.693,A -85,B 0,C 180,E1 -19814.273,E2 -19814.273} C_VEL
LIN {X 0,Y 227.992,Z 157.7,A -85,B 0,C 180,E1 -19817.954,E2 -19817.954} C_VEL
LIN {X 0,Y 227.924,Z 157.709,A -85,B 0,C 180,E1 -19822.324,E2 -19822.324} C_VEL
LIN {X 0,Y 227.925,Z 157.709,A -85,B 0,C 180,E1 -19826.592,E2 -19826.592} C_VEL
LIN {X 0,Y 227.875,Z 157.727,A -85,B 0,C 180,E1 -19830.281,E2 -19830.281} C_VEL
LIN {X 0,Y 227.87,Z 157.751,A -85,B 0,C 180,E1 -19831.752,E2 -19831.752} C_VEL
LIN {X 0,Y 228.136,Z 158.867,A -85,B 0,C 180,E1 -19832.361,E2 -19832.361} C_VEL
LIN {X 0,Y 229.555,Z 161.459,A -85,B 0,C 180,E1 -19833.057,E2 -19833.057} C_VEL
LIN {X 0,Y 232.834,Z 165.202,A -85,B 0,C 180,E1 -19834.469,E2 -19834.469} C_VEL
LIN {X 0,Y 236.568,Z 170.429,A -85,B 0,C 180,E1 -19836.021,E2 -19836.021} C_VEL
LIN {X 0,Y 241.707,Z 178.286,A -85,B 0,C 180,E1 -19838.025,E2 -19838.025} C_VEL
LIN {X 0,Y 245.53,Z 184.427,A -85,B 0,C 180,E1 -19839.422,E2 -19839.422} C_VEL
LIN {X 0,Y 252.236,Z 195.632,A -85,B 0,C 180,E1 -19841.7,E2 -19841.7} C_VEL
LIN {X 0,Y 259.273,Z 208.954,A -85,B 0,C 180,E1 -19843.928,E2 -19843.928} C_VEL
LIN {X 0,Y 265.793,Z 222.87,A -85,B 0,C 180,E1 -19845.874,E2 -19845.874} C_VEL
LIN {X 0,Y 269.473,Z 231.796,A -85,B 0,C 180,E1 -19846.942,E2 -19846.942} C_VEL
LIN {X 0,Y 264.319,Z 326.52,A -85,B 0,C 180,E1 -19849.35,E2 -19849.35} C_VEL
LIN {X 0,Y 262.491,Z 342.697,A -85,B 0,C 180,E1 -19850.015,E2 -19850.015} C_VEL
LIN {X 0,Y 259.964,Z 357.955,A -85,B 0,C 180,E1 -19850.932,E2 -19850.932} C_VEL
LIN {X 0,Y 257.136,Z 371.697,A -85,B 0,C 180,E1 -19852.05,E2 -19852.05} C_VEL
LIN {X 0,Y 254.014,Z 384.606,A -85,B 0,C 180,E1 -19853.41,E2 -19853.41} C_VEL
LIN {X 0,Y 250.381,Z 397.587,A -85,B 0,C 180,E1 -19855.116,E2 -19855.116} C_VEL
LIN {X 0,Y 246.633,Z 409.154,A -85,B 0,C 180,E1 -19856.976,E2 -19856.976} C_VEL
LIN {X 0,Y 242.922,Z 419.929,A -85,B 0,C 180,E1 -19859.101,E2 -19859.101} C_VEL
LIN {X 0,Y 239.373,Z 429.906,A -85,B 0,C 180,E1 -19861.504,E2 -19861.504} C_VEL
LIN {X 0,Y 235.833,Z 439.676,A -85,B 0,C 180,E1 -19864.398,E2 -19864.398} C_VEL
LIN {X 0,Y 232.635,Z 447.827,A -85,B 0,C 180,E1 -19867.345,E2 -19867.345} C_VEL
LIN {X 0,Y 230.134,Z 454.575,A -85,B 0,C 180,E1 -19870.371,E2 -19870.371} C_VEL
LIN {X 0,Y 228.04,Z 460.814,A -85,B 0,C 180,E1 -19873.896,E2 -19873.896} C_VEL
LIN {X 0,Y 226.566,Z 465.643,A -85,B 0,C 180,E1 -19877.459,E2 -19877.459} C_VEL
LIN {X 0,Y 225.809,Z 469.189,A -85,B 0,C 180,E1 -19881.047,E2 -19881.047} C_VEL
LIN {X 0,Y 225.561,Z 471.526,A -85,B 0,C 180,E1 -19884.636,E2 -19884.636} C_VEL
LIN {X 0,Y 225.633,Z 472.704,A -85,B 0,C 180,E1 -19888.215,E2 -19888.215} C_VEL
LIN {X 0,Y 225.713,Z 472.86,A -85,B 0,C 180,E1 -19890,E2 -19890} C_VEL
LIN {X 0,Y 225.548,Z 472.243,A -85,B 0,C 180,E1 -19893.573,E2 -19893.573} C_VEL
LIN {X 0,Y 225.617,Z 470.472,A -85,B 0,C 180,E1 -19897.158,E2 -19897.158} C_VEL
LIN {X 0,Y 226.129,Z 467.526,A -85,B 0,C 180,E1 -19900.747,E2 -19900.747} C_VEL
LIN {X 0,Y 227.244,Z 463.34,A -85,B 0,C 180,E1 -19904.325,E2 -19904.325} C_VEL
LIN {X 0,Y 228.885,Z 457.799,A -85,B 0,C 180,E1 -19907.882,E2 -19907.882} C_VEL
LIN {X 0,Y 231.442,Z 450.766,A -85,B 0,C 180,E1 -19911.37,E2 -19911.37} C_VEL
LIN {X 0,Y 234.321,Z 443.25,A -85,B 0,C 180,E1 -19914.356,E2 -19914.356} C_VEL
LIN {X 0,Y 237.459,Z 434.788,A -85,B 0,C 180,E1 -19917.098,E2 -19917.098} C_VEL
LIN {X 0,Y 241.044,Z 424.953,A -85,B 0,C 180,E1 -19919.713,E2 -19919.713} C_VEL
LIN {X 0,Y 244.879,Z 414.074,A -85,B 0,C 180,E1 -19922.07,E2 -19922.07} C_VEL
LIN {X 0,Y 248.798,Z 402.205,A -85,B 0,C 180,E1 -19924.155,E2 -19924.155} C_VEL
LIN {X 0,Y 252.701,Z 389.31,A -85,B 0,C 180,E1 -19925.967,E2 -19925.967} C_VEL
LIN {X 0,Y 255.876,Z 376.653,A -85,B 0,C 180,E1 -19927.423,E2 -19927.423} C_VEL
LIN {X 0,Y 258.843,Z 363.135,A -85,B 0,C 180,E1 -19928.645,E2 -19928.645} C_VEL
LIN {X 0,Y 261.572,Z 348.169,A -85,B 0,C 180,E1 -19929.652,E2 -19929.652} C_VEL
LIN {X 0,Y 263.524,Z 333.61,A -85,B 0,C 180,E1 -19930.358,E2 -19930.358} C_VEL
LIN {X 0,Y 264.792,Z 317.44,A -85,B 0,C 180,E1 -19930.875,E2 -19930.875} C_VEL
LIN {X 0,Y 269.341,Z 232.137,A -85,B 0,C 180,E1 -19933.016,E2 -19933.016} C_VEL
LIN {X 0,Y 268.743,Z 230.088,A -85,B 0,C 180,E1 -19933.208,E2 -19933.208} C_VEL
LIN {X 0,Y 263.07,Z 216.917,A -85,B 0,C 180,E1 -19934.864,E2 -19934.864} C_VEL
LIN {X 0,Y 255.629,Z 201.97,A -85,B 0,C 180,E1 -19937.134,E2 -19937.134} C_VEL
LIN {X 0,Y 248.955,Z 190.088,A -85,B 0,C 180,E1 -19939.312,E2 -19939.312} C_VEL
LIN {X 0,Y 242.743,Z 179.958,A -85,B 0,C 180,E1 -19941.502,E2 -19941.502} C_VEL
LIN {X 0,Y 239.439,Z 174.876,A -85,B 0,C 180,E1 -19942.744,E2 -19942.744} C_VEL
LIN {X 0,Y 235.917,Z 169.625,A -85,B 0,C 180,E1 -19944.139,E2 -19944.139} C_VEL
LIN {X 0,Y 231.877,Z 164.088,A -85,B 0,C 180,E1 -19945.829,E2 -19945.829} C_VEL
LIN {X 0,Y 228.638,Z 160.043,A -85,B 0,C 180,E1 -19947.262,E2 -19947.262} C_VEL
LIN {X 0,Y 228.061,Z 158.577,A -85,B 0,C 180,E1 -19947.627,E2 -19947.627} C_VEL
LIN {X 0,Y 227.896,Z 157.718,A -85,B 0,C 180,E1 -19948.252,E2 -19948.252} C_VEL
LIN {X 0,Y 227.888,Z 157.716,A -85,B 0,C 180,E1 -19952.445,E2 -19952.445} C_VEL
LIN {X 0,Y 227.916,Z 157.712,A -85,B 0,C 180,E1 -19956.368,E2 -19956.368} C_VEL
LIN {X 0,Y 227.944,Z 157.707,A -85,B 0,C 180,E1 -19960.175,E2 -19960.175} C_VEL
LIN {X 0,Y 228.06,Z 157.692,A -85,B 0,C 180,E1 -19963.898,E2 -19963.898} C_VEL
LIN {X 0,Y 228.065,Z 157.69,A -85,B 0,C 180,E1 -19967.543,E2 -19967.543} C_VEL
LIN {X 0,Y 228.254,Z 157.667,A -85,B 0,C 180,E1 -19971.144,E2 -19971.144} C_VEL
LIN {X 0,Y 228.304,Z 157.666,A -85,B 0,C 180,E1 -19972.927,E2 -19972.927} C_VEL
LIN {X 0,Y 228.55,Z 157.643,A -85,B 0,C 180,E1 -19978.238,E2 -19978.238} C_VEL
LIN {X 0,Y 228.539,Z 157.64,A -85,B 0,C 180,E1 -19981.762,E2 -19981.762} C_VEL
LIN {X 0,Y 228.303,Z 157.672,A -85,B 0,C 180,E1 -19987.073,E2 -19987.073} C_VEL
LIN {X 0,Y 228.142,Z 157.691,A -85,B 0,C 180,E1 -19990.652,E2 -19990.652} C_VEL
LIN {X 0,Y 228.016,Z 157.702,A -85,B 0,C 180,E1 -19996.105,E2 -19996.105} C_VEL
LIN {X 0,Y 227.918,Z 157.717,A -85,B 0,C 180,E1 -19999.828,E2 -19999.828} C_VEL
LIN {X 0,Y 227.896,Z 157.719,A -85,B 0,C 180,E1 -20003.635,E2 -20003.635} C_VEL
LIN {X 0,Y 227.856,Z 157.694,A -85,B 0,C 180,E1 -20007.559,E2 -20007.559} C_VEL
LIN {X 0,Y 227.857,Z 157.72,A -85,B 0,C 180,E1 -20011.624,E2 -20011.624} C_VEL
LIN {X 0,Y 227.904,Z 157.729,A -85,B 0,C 180,E1 -20012.759,E2 -20012.759} C_VEL
LIN {X 0,Y 228.673,Z 160.185,A -85,B 0,C 180,E1 -20013.199,E2 -20013.199} C_VEL
LIN {X 0,Y 230.603,Z 162.48,A -85,B 0,C 180,E1 -20014.057,E2 -20014.057} C_VEL
LIN {X 0,Y 231.981,Z 163.467,A -85,B 0,C 180,E1 -20014.614,E2 -20014.614} C_VEL
LIN {X 0,Y 233.956,Z 166.706,A -85,B 0,C 180,E1 -20015.484,E2 -20015.484} C_VEL
LIN {X 0,Y 235.979,Z 168.783,A -85,B 0,C 180,E1 -20016.278,E2 -20016.278} C_VEL
LIN {X 0,Y 238.517,Z 172.315,A -85,B 0,C 180,E1 -20017.28,E2 -20017.28} C_VEL
LIN {X 0,Y 240.399,Z 174.909,A -85,B 0,C 180,E1 -20017.994,E2 -20017.994} C_VEL
LIN {X 0,Y 243.427,Z 178.968,A -85,B 0,C 180,E1 -20019.092,E2 -20019.092} C_VEL
LIN {X 0,Y 249.15,Z 187.08,A -85,B 0,C 180,E1 -20021.049,E2 -20021.049} C_VEL
LIN {X 0,Y 256.116,Z 197.712,A -85,B 0,C 180,E1 -20023.25,E2 -20023.25} C_VEL
LIN {X 0,Y 262.388,Z 208.315,A -85,B 0,C 180,E1 -20025.102,E2 -20025.102} C_VEL
LIN {X 0,Y 268.746,Z 221.805,A -85,B 0,C 180,E1 -20026.935,E2 -20026.935} C_VEL
LIN {X 0,Y 269.679,Z 223.955,A -85,B 0,C 180,E1 -20027.198,E2 -20027.198} C_VEL
LIN {X 0,Y 264.775,Z 314.425,A -85,B 0,C 180,E1 -20029.497,E2 -20029.497} C_VEL
LIN {X 0,Y 263.114,Z 330.093,A -85,B 0,C 180,E1 -20030.129,E2 -20030.129} C_VEL
LIN {X 0,Y 260.872,Z 345.705,A -85,B 0,C 180,E1 -20031.094,E2 -20031.094} C_VEL
LIN {X 0,Y 258.273,Z 359.496,A -85,B 0,C 180,E1 -20032.244,E2 -20032.244} C_VEL
LIN {X 0,Y 255.194,Z 373.07,A -85,B 0,C 180,E1 -20033.693,E2 -20033.693} C_VEL
LIN {X 0,Y 251.393,Z 386.827,A -85,B 0,C 180,E1 -20035.52,E2 -20035.52} C_VEL
LIN {X 0,Y 247.489,Z 399.238,A -85,B 0,C 180,E1 -20037.588,E2 -20037.588} C_VEL
LIN {X 0,Y 243.324,Z 411.171,A -85,B 0,C 180,E1 -20040.055,E2 -20040.055} C_VEL
LIN {X 0,Y 239.921,Z 420.735,A -85,B 0,C 180,E1 -20042.525,E2 -20042.525} C_VEL
LIN {X 0,Y 236.376,Z 429.921,A -85,B 0,C 180,E1 -20045.402,E2 -20045.402} C_VEL
LIN {X 0,Y 233.3,Z 437.555,A -85,B 0,C 180,E1 -20048.345,E2 -20048.345} C_VEL
LIN {X 0,Y 230.845,Z 443.884,A -85,B 0,C 180,E1 -20051.357,E2 -20051.357} C_VEL
LIN {X 0,Y 228.725,Z 449.691,A -85,B 0,C 180,E1 -20054.86,E2 -20054.86} C_VEL
LIN {X 0,Y 227.543,Z 453.128,A -85,B 0,C 180,E1 -20057.514,E2 -20057.514} C_VEL
LIN {X 0,Y 226.521,Z 456.602,A -85,B 0,C 180,E1 -20061.076,E2 -20061.076} C_VEL
LIN {X 0,Y 225.923,Z 458.897,A -85,B 0,C 180,E1 -20064.645,E2 -20064.645} C_VEL
LIN {X 0,Y 225.738,Z 460.063,A -85,B 0,C 180,E1 -20068.216,E2 -20068.216} C_VEL
LIN {X 0,Y 225.738,Z 460.076,A -85,B 0,C 180,E1 -20071.784,E2 -20071.784} C_VEL
LIN {X 0,Y 225.918,Z 458.92,A -85,B 0,C 180,E1 -20075.449,E2 -20075.449} C_VEL
LIN {X 0,Y 226.495,Z 456.715,A -85,B 0,C 180,E1 -20078.925,E2 -20078.925} C_VEL
LIN {X 0,Y 227.496,Z 453.285,A -85,B 0,C 180,E1 -20082.489,E2 -20082.489} C_VEL
LIN {X 0,Y 229.208,Z 448.581,A -85,B 0,C 180,E1 -20086.019,E2 -20086.019} C_VEL
LIN {X 0,Y 231.449,Z 442.486,A -85,B 0,C 180,E1 -20089.513,E2 -20089.513} C_VEL
LIN {X 0,Y 234.457,Z 434.803,A -85,B 0,C 180,E1 -20092.935,E2 -20092.935} C_VEL
LIN {X 0,Y 237.729,Z 426.607,A -85,B 0,C 180,E1 -20095.853,E2 -20095.853} C_VEL
LIN {X 0,Y 241.58,Z 416.725,A -85,B 0,C 180,E1 -20098.687,E2 -20098.687} C_VEL
LIN {X 0,Y 245.044,Z 406.601,A -85,B 0,C 180,E1 -20101.081,E2 -20101.081} C_VEL
LIN {X 0,Y 249.151,Z 394.529,A -85,B 0,C 180,E1 -20103.371,E2 -20103.371} C_VEL
LIN {X 0,Y 252.708,Z 382.424,A -85,B 0,C 180,E1 -20105.245,E2 -20105.245} C_VEL
LIN {X 0,Y 256.169,Z 369.261,A -85,B 0,C 180,E1 -20106.88,E2 -20106.88} C_VEL
LIN {X 0,Y 259.15,Z 355.541,A -85,B 0,C 180,E1 -20108.241,E2 -20108.241} C_VEL
LIN {X 0,Y 261.756,Z 340.708,A -85,B 0,C 180,E1 -20109.37,E2 -20109.37} C_VEL
LIN {X 0,Y 263.799,Z 325.779,A -85,B 0,C 180,E1 -20110.183,E2 -20110.183} C_VEL
LIN {X 0,Y 265.161,Z 310.361,A -85,B 0,C 180,E1 -20110.744,E2 -20110.744} C_VEL
LIN {X 0,Y 269.241,Z 233.972,A -85,B 0,C 180,E1 -20112.677,E2 -20112.677} C_VEL
LIN {X 0,Y 269.74,Z 223.905,A -85,B 0,C 180,E1 -20112.938,E2 -20112.938} C_VEL
LIN {X 0,Y 263.379,Z 210.169,A -85,B 0,C 180,E1 -20114.763,E2 -20114.763} C_VEL
LIN {X 0,Y 259.24,Z 202.684,A -85,B 0,C 180,E1 -20115.976,E2 -20115.976} C_VEL
LIN {X 0,Y 250.827,Z 189.423,A -85,B 0,C 180,E1 -20118.575,E2 -20118.575} C_VEL
LIN {X 0,Y 244.862,Z 180.862,A -85,B 0,C 180,E1 -20120.58,E2 -20120.58} C_VEL
LIN {X 0,Y 241.32,Z 176.152,A -85,B 0,C 180,E1 -20121.844,E2 -20121.844} C_VEL
LIN {X 0,Y 238.631,Z 172.43,A -85,B 0,C 180,E1 -20122.861,E2 -20122.861} C_VEL
LIN {X 0,Y 236.046,Z 168.881,A -85,B 0,C 180,E1 -20123.882,E2 -20123.882} C_VEL
LIN {X 0,Y 232.804,Z 165.125,A -85,B 0,C 180,E1 -20125.197,E2 -20125.197} C_VEL
LIN {X 0,Y 231.877,Z 163.242,A -85,B 0,C 180,E1 -20125.632,E2 -20125.632} C_VEL
LIN {X 0,Y 229.511,Z 161.404,A -85,B 0,C 180,E1 -20126.614,E2 -20126.614} C_VEL
LIN {X 0,Y 228.202,Z 159.002,A -85,B 0,C 180,E1 -20127.256,E2 -20127.256} C_VEL
LIN {X 0,Y 227.913,Z 157.69,A -85,B 0,C 180,E1 -20127.472,E2 -20127.472} C_VEL
LIN {X 0,Y 227.873,Z 157.699,A -85,B 0,C 180,E1 -20130.431,E2 -20130.431} C_VEL
LIN {X 0,Y 227.873,Z 157.716,A -85,B 0,C 180,E1 -20134.419,E2 -20134.419} C_VEL
LIN {X 0,Y 227.921,Z 157.709,A -85,B 0,C 180,E1 -20138.283,E2 -20138.283} C_VEL
LIN {X 0,Y 228.018,Z 157.708,A -85,B 0,C 180,E1 -20143.895,E2 -20143.895} C_VEL
LIN {X 0,Y 228.144,Z 157.686,A -85,B 0,C 180,E1 -20149.349,E2 -20149.349} C_VEL
LIN {X 0,Y 228.302,Z 157.672,A -85,B 0,C 180,E1 -20152.927,E2 -20152.927} C_VEL
LIN {X 0,Y 228.538,Z 157.641,A -85,B 0,C 180,E1 -20158.238,E2 -20158.238} C_VEL
LIN {X 0,Y 228.569,Z 157.624,A -85,B 0,C 180,E1 -20159.872,E2 -20159.872} C_VEL
LIN {X 0,Y 227.964,Z 157.708,A -85,B 0,C 180,E1 -20161.338,E2 -20161.338} C_VEL
LIN {X 0,Y 226.366,Z 157.914,A -85,B 0,C 180,E1 -20162.776,E2 -20162.776} C_VEL
LIN {X 0,Y 222.478,Z 158.406,A -85,B 0,C 180,E1 -20165.672,E2 -20165.672} C_VEL
LIN {X 0,Y 221.331,Z 158.543,A -85,B 0,C 180,E1 -20167.189,E2 -20167.189} C_VEL
LIN {X 0,Y 221.216,Z 158.55,A -85,B 0,C 180,E1 -20167.705,E2 -20167.705} C_VEL
LIN {X 0,Y 221.068,Z 158.572,A -85,B 0,C 180,E1 -20170.996,E2 -20170.996} C_VEL
LIN {X 0,Y 220.993,Z 158.582,A -85,B 0,C 180,E1 -20176.631,E2 -20176.631} C_VEL
LIN {X 0,Y 220.884,Z 158.6,A -85,B 0,C 180,E1 -20180.487,E2 -20180.487} C_VEL
LIN {X 0,Y 220.852,Z 158.604,A -85,B 0,C 180,E1 -20184.437,E2 -20184.437} C_VEL
LIN {X 0,Y 220.807,Z 158.607,A -85,B 0,C 180,E1 -20188.518,E2 -20188.518} C_VEL
LIN {X 0,Y 220.813,Z 158.621,A -85,B 0,C 180,E1 -20189.232,E2 -20189.232} C_VEL
LIN {X 0,Y 221.635,Z 161.104,A -85,B 0,C 180,E1 -20189.766,E2 -20189.766} C_VEL
LIN {X 0,Y 223.511,Z 163.336,A -85,B 0,C 180,E1 -20190.727,E2 -20190.727} C_VEL
LIN {X 0,Y 225.209,Z 164.555,A -85,B 0,C 180,E1 -20191.514,E2 -20191.514} C_VEL
LIN {X 0,Y 227.158,Z 167.722,A -85,B 0,C 180,E1 -20192.484,E2 -20192.484} C_VEL
LIN {X 0,Y 230.461,Z 171.771,A -85,B 0,C 180,E1 -20193.965,E2 -20193.965} C_VEL
LIN {X 0,Y 234.843,Z 178.285,A -85,B 0,C 180,E1 -20195.844,E2 -20195.844} C_VEL
LIN {X 0,Y 238.324,Z 183.585,A -85,B 0,C 180,E1 -20197.238,E2 -20197.238} C_VEL
LIN {X 0,Y 244.875,Z 194.414,A -85,B 0,C 180,E1 -20199.686,E2 -20199.686} C_VEL
LIN {X 0,Y 251.417,Z 206.182,A -85,B 0,C 180,E1 -20201.933,E2 -20201.933} C_VEL
LIN {X 0,Y 257.773,Z 219.003,A -85,B 0,C 180,E1 -20203.978,E2 -20203.978} C_VEL
LIN {X 0,Y 263.985,Z 233.465,A -85,B 0,C 180,E1 -20205.887,E2 -20205.887} C_VEL
LIN {X 0,Y 264.15,Z 235.357,A -85,B 0,C 180,E1 -20205.992,E2 -20205.992} C_VEL
LIN {X 0,Y 258.984,Z 326.338,A -85,B 0,C 180,E1 -20208.329,E2 -20208.329} C_VEL
LIN {X 0,Y 257.101,Z 342.507,A -85,B 0,C 180,E1 -20209,E2 -20209} C_VEL
LIN {X 0,Y 254.492,Z 357.763,A -85,B 0,C 180,E1 -20209.924,E2 -20209.924} C_VEL
LIN {X 0,Y 251.545,Z 371.503,A -85,B 0,C 180,E1 -20211.05,E2 -20211.05} C_VEL
LIN {X 0,Y 248.168,Z 385.011,A -85,B 0,C 180,E1 -20212.499,E2 -20212.499} C_VEL
LIN {X 0,Y 244.179,Z 398.685,A -85,B 0,C 180,E1 -20214.349,E2 -20214.349} C_VEL
LIN {X 0,Y 240.328,Z 410.031,A -85,B 0,C 180,E1 -20216.246,E2 -20216.246} C_VEL
LIN {X 0,Y 236.15,Z 421.522,A -85,B 0,C 180,E1 -20218.613,E2 -20218.613} C_VEL
LIN {X 0,Y 232.528,Z 431.201,A -85,B 0,C 180,E1 -20221.08,E2 -20221.08} C_VEL
LIN {X 0,Y 228.875,Z 440.716,A -85,B 0,C 180,E1 -20224.051,E2 -20224.051} C_VEL
LIN {X 0,Y 225.601,Z 448.643,A -85,B 0,C 180,E1 -20227.082,E2 -20227.082} C_VEL
LIN {X 0,Y 222.769,Z 456.054,A -85,B 0,C 180,E1 -20230.655,E2 -20230.655} C_VEL
LIN {X 0,Y 220.706,Z 461.94,A -85,B 0,C 180,E1 -20234.296,E2 -20234.296} C_VEL
LIN {X 0,Y 219.583,Z 465.444,A -85,B 0,C 180,E1 -20237.053,E2 -20237.053} C_VEL
LIN {X 0,Y 218.755,Z 468.989,A -85,B 0,C 180,E1 -20240.756,E2 -20240.756} C_VEL
LIN {X 0,Y 218.476,Z 471.327,A -85,B 0,C 180,E1 -20244.462,E2 -20244.462} C_VEL
LIN {X 0,Y 218.529,Z 472.505,A -85,B 0,C 180,E1 -20248.157,E2 -20248.157} C_VEL
LIN {X 0,Y 218.628,Z 472.662,A -85,B 0,C 180,E1 -20250,E2 -20250} C_VEL
LIN {X 0,Y 218.449,Z 472.044,A -85,B 0,C 180,E1 -20253.689,E2 -20253.689} C_VEL
LIN {X 0,Y 218.552,Z 470.272,A -85,B 0,C 180,E1 -20257.39,E2 -20257.39} C_VEL
LIN {X 0,Y 219.111,Z 467.325,A -85,B 0,C 180,E1 -20261.096,E2 -20261.096} C_VEL
LIN {X 0,Y 220.313,Z 463.138,A -85,B 0,C 180,E1 -20264.785,E2 -20264.785} C_VEL
LIN {X 0,Y 222.096,Z 457.597,A -85,B 0,C 180,E1 -20268.448,E2 -20268.448} C_VEL
LIN {X 0,Y 224.789,Z 450.564,A -85,B 0,C 180,E1 -20272.035,E2 -20272.035} C_VEL
LIN {X 0,Y 227.834,Z 443.049,A -85,B 0,C 180,E1 -20275.097,E2 -20275.097} C_VEL
LIN {X 0,Y 231.264,Z 434.127,A -85,B 0,C 180,E1 -20278.052,E2 -20278.052} C_VEL
LIN {X 0,Y 235.476,Z 423.108,A -85,B 0,C 180,E1 -20280.987,E2 -20280.987} C_VEL
LIN {X 0,Y 239.896,Z 410.88,A -85,B 0,C 180,E1 -20283.571,E2 -20283.571} C_VEL
LIN {X 0,Y 244.153,Z 398.418,A -85,B 0,C 180,E1 -20285.655,E2 -20285.655} C_VEL
LIN {X 0,Y 247.854,Z 385.841,A -85,B 0,C 180,E1 -20287.364,E2 -20287.364} C_VEL
LIN {X 0,Y 251.537,Z 371.069,A -85,B 0,C 180,E1 -20288.951,E2 -20288.951} C_VEL
LIN {X 0,Y 254.703,Z 356.008,A -85,B 0,C 180,E1 -20290.165,E2 -20290.165} C_VEL
LIN {X 0,Y 257.234,Z 340.913,A -85,B 0,C 180,E1 -20291.039,E2 -20291.039} C_VEL
LIN {X 0,Y 258.967,Z 325.037,A -85,B 0,C 180,E1 -20291.675,E2 -20291.675} C_VEL
LIN {X 0,Y 264.049,Z 233.808,A -85,B 0,C 180,E1 -20294.027,E2 -20294.027} C_VEL
LIN {X 0,Y 258.68,Z 221.141,A -85,B 0,C 180,E1 -20295.668,E2 -20295.668} C_VEL
LIN {X 0,Y 251.526,Z 206.486,A -85,B 0,C 180,E1 -20297.955,E2 -20297.955} C_VEL
LIN {X 0,Y 245.315,Z 195.222,A -85,B 0,C 180,E1 -20300.075,E2 -20300.075} C_VEL
LIN {X 0,Y 239.129,Z 184.929,A -85,B 0,C 180,E1 -20302.356,E2 -20302.356} C_VEL
LIN {X 0,Y 236.166,Z 180.328,A -85,B 0,C 180,E1 -20303.52,E2 -20303.52} C_VEL
LIN {X 0,Y 232.762,Z 175.188,A -85,B 0,C 180,E1 -20304.927,E2 -20304.927} C_VEL
LIN {X 0,Y 229.076,Z 169.946,A -85,B 0,C 180,E1 -20306.541,E2 -20306.541} C_VEL
LIN {X 0,Y 225.796,Z 165.781,A -85,B 0,C 180,E1 -20308.053,E2 -20308.053} C_VEL
LIN {X 0,Y 225.029,Z 164.227,A -85,B 0,C 180,E1 -20308.458,E2 -20308.458} C_VEL
LIN {X 0,Y 222.502,Z 162.316,A -85,B 0,C 180,E1 -20309.644,E2 -20309.644} C_VEL
LIN {X 0,Y 221.2,Z 160.006,A -85,B 0,C 180,E1 -20310.366,E2 -20310.366} C_VEL
LIN {X 0,Y 220.878,Z 158.588,A -85,B 0,C 180,E1 -20310.646,E2 -20310.646} C_VEL
LIN {X 0,Y 220.897,Z 158.586,A -85,B 0,C 180,E1 -20313.55,E2 -20313.55} C_VEL
LIN {X 0,Y 220.88,Z 158.593,A -85,B 0,C 180,E1 -20317.554,E2 -20317.554} C_VEL
LIN {X 0,Y 220.986,Z 158.578,A -85,B 0,C 180,E1 -20322.571,E2 -20322.571} C_VEL
LIN {X 0,Y 221.006,Z 158.57,A -85,B 0,C 180,E1 -20327.138,E2 -20327.138} C_VEL
LIN {X 0,Y 221.195,Z 158.548,A -85,B 0,C 180,E1 -20330.859,E2 -20330.859} C_VEL
LIN {X 0,Y 221.123,Z 158.562,A -85,B 0,C 180,E1 -20334.529,E2 -20334.529} C_VEL
LIN {X 0,Y 221.508,Z 158.52,A -85,B 0,C 180,E1 -20338.182,E2 -20338.182} C_VEL
LIN {X 0,Y 221.472,Z 158.521,A -85,B 0,C 180,E1 -20341.819,E2 -20341.819} C_VEL
LIN {X 0,Y 221.24,Z 158.55,A -85,B 0,C 180,E1 -20347.3,E2 -20347.3} C_VEL
LIN {X 0,Y 221.062,Z 158.574,A -85,B 0,C 180,E1 -20350.997,E2 -20350.997} C_VEL
LIN {X 0,Y 220.976,Z 158.575,A -85,B 0,C 180,E1 -20356.633,E2 -20356.633} C_VEL
LIN {X 0,Y 220.873,Z 158.589,A -85,B 0,C 180,E1 -20360.488,E2 -20360.488} C_VEL
LIN {X 0,Y 220.848,Z 158.579,A -85,B 0,C 180,E1 -20364.437,E2 -20364.437} C_VEL
LIN {X 0,Y 220.805,Z 158.585,A -85,B 0,C 180,E1 -20368.518,E2 -20368.518} C_VEL
LIN {X 0,Y 220.836,Z 158.628,A -85,B 0,C 180,E1 -20369.819,E2 -20369.819} C_VEL
LIN {X 0,Y 221.661,Z 161.16,A -85,B 0,C 180,E1 -20370.353,E2 -20370.353} C_VEL
LIN {X 0,Y 223.448,Z 163.291,A -85,B 0,C 180,E1 -20371.263,E2 -20371.263} C_VEL
LIN {X 0,Y 225.161,Z 164.438,A -85,B 0,C 180,E1 -20372.048,E2 -20372.048} C_VEL
LIN {X 0,Y 226.896,Z 167.448,A -85,B 0,C 180,E1 -20372.92,E2 -20372.92} C_VEL
LIN {X 0,Y 229.378,Z 169.951,A -85,B 0,C 180,E1 -20374.012,E2 -20374.012} C_VEL
LIN {X 0,Y 231.968,Z 173.517,A -85,B 0,C 180,E1 -20375.145,E2 -20375.145} C_VEL
LIN {X 0,Y 233.353,Z 175.212,A -85,B 0,C 180,E1 -20375.718,E2 -20375.718} C_VEL
LIN {X 0,Y 237.112,Z 180.299,A -85,B 0,C 180,E1 -20377.224,E2 -20377.224} C_VEL
LIN {X 0,Y 243.062,Z 188.576,A -85,B 0,C 180,E1 -20379.427,E2 -20379.427} C_VEL
LIN {X 0,Y 250.488,Z 199.834,A -85,B 0,C 180,E1 -20381.942,E2 -20381.942} C_VEL
LIN {X 0,Y 257.462,Z 211.433,A -85,B 0,C 180,E1 -20384.114,E2 -20384.114} C_VEL
LIN {X 0,Y 263.475,Z 224.212,A -85,B 0,C 180,E1 -20385.935,E2 -20385.935} C_VEL
LIN {X 0,Y 264.402,Z 226.296,A -85,B 0,C 180,E1 -20386.208,E2 -20386.208} C_VEL
LIN {X 0,Y 259.426,Z 314.644,A -85,B 0,C 180,E1 -20388.481,E2 -20388.481} C_VEL
LIN {X 0,Y 257.701,Z 330.304,A -85,B 0,C 180,E1 -20389.116,E2 -20389.116} C_VEL
LIN {X 0,Y 255.383,Z 345.912,A -85,B 0,C 180,E1 -20390.093,E2 -20390.093} C_VEL
LIN {X 0,Y 252.549,Z 360.431,A -85,B 0,C 180,E1 -20391.326,E2 -20391.326} C_VEL
LIN {X 0,Y 249.122,Z 374.825,A -85,B 0,C 180,E1 -20392.914,E2 -20392.914} C_VEL
LIN {X 0,Y 245.195,Z 388.274,A -85,B 0,C 180,E1 -20394.771,E2 -20394.771} C_VEL
LIN {X 0,Y 241.149,Z 400.48,A -85,B 0,C 180,E1 -20396.876,E2 -20396.876} C_VEL
LIN {X 0,Y 236.953,Z 411.952,A -85,B 0,C 180,E1 -20399.332,E2 -20399.332} C_VEL
LIN {X 0,Y 233.643,Z 420.936,A -85,B 0,C 180,E1 -20401.721,E2 -20401.721} C_VEL
LIN {X 0,Y 229.895,Z 430.123,A -85,B 0,C 180,E1 -20404.66,E2 -20404.66} C_VEL
LIN {X 0,Y 226.675,Z 437.757,A -85,B 0,C 180,E1 -20407.678,E2 -20407.678} C_VEL
LIN {X 0,Y 224.088,Z 444.085,A -85,B 0,C 180,E1 -20410.773,E2 -20410.773} C_VEL
LIN {X 0,Y 221.843,Z 449.892,A -85,B 0,C 180,E1 -20414.379,E2 -20414.379} C_VEL
LIN {X 0,Y 220.581,Z 453.328,A -85,B 0,C 180,E1 -20417.113,E2 -20417.113} C_VEL
LIN {X 0,Y 219.507,Z 456.802,A -85,B 0,C 180,E1 -20420.788,E2 -20420.788} C_VEL
LIN {X 0,Y 218.838,Z 459.154,A -85,B 0,C 180,E1 -20424.606,E2 -20424.606} C_VEL
LIN {X 0,Y 218.656,Z 460.262,A -85,B 0,C 180,E1 -20428.158,E2 -20428.158} C_VEL
LIN {X 0,Y 218.656,Z 460.274,A -85,B 0,C 180,E1 -20431.842,E2 -20431.842} C_VEL
LIN {X 0,Y 218.847,Z 459.159,A -85,B 0,C 180,E1 -20435.529,E2 -20435.529} C_VEL
LIN {X 0,Y 219.46,Z 456.914,A -85,B 0,C 180,E1 -20439.214,E2 -20439.214} C_VEL
LIN {X 0,Y 220.542,Z 453.483,A -85,B 0,C 180,E1 -20442.889,E2 -20442.889} C_VEL
LIN {X 0,Y 222.373,Z 448.779,A -85,B 0,C 180,E1 -20446.526,E2 -20446.526} C_VEL
LIN {X 0,Y 224.734,Z 442.684,A -85,B 0,C 180,E1 -20450.121,E2 -20450.121} C_VEL
LIN {X 0,Y 227.913,Z 435.001,A -85,B 0,C 180,E1 -20453.633,E2 -20453.633} C_VEL
LIN {X 0,Y 231.303,Z 426.805,A -85,B 0,C 180,E1 -20456.626,E2 -20456.626} C_VEL
LIN {X 0,Y 235.346,Z 416.922,A -85,B 0,C 180,E1 -20459.52,E2 -20459.52} C_VEL
LIN {X 0,Y 238.971,Z 406.797,A -85,B 0,C 180,E1 -20461.963,E2 -20461.963} C_VEL
LIN {X 0,Y 243.241,Z 394.724,A -85,B 0,C 180,E1 -20464.293,E2 -20464.293} C_VEL
LIN {X 0,Y 246.544,Z 383.905,A -85,B 0,C 180,E1 -20466.011,E2 -20466.011} C_VEL
LIN {X 0,Y 250.143,Z 371.03,A -85,B 0,C 180,E1 -20467.668,E2 -20467.668} C_VEL
LIN {X 0,Y 253.311,Z 357.077,A -85,B 0,C 180,E1 -20469.116,E2 -20469.116} C_VEL
LIN {X 0,Y 256.105,Z 342.196,A -85,B 0,C 180,E1 -20470.286,E2 -20470.286} C_VEL
LIN {X 0,Y 258.269,Z 326.881,A -85,B 0,C 180,E1 -20471.162,E2 -20471.162} C_VEL
LIN {X 0,Y 259.707,Z 312.043,A -85,B 0,C 180,E1 -20471.724,E2 -20471.724} C_VEL
LIN {X 0,Y 263.909,Z 237.636,A -85,B 0,C 180,E1 -20473.625,E2 -20473.625} C_VEL
LIN {X 0,Y 264.467,Z 226.273,A -85,B 0,C 180,E1 -20473.929,E2 -20473.929} C_VEL
LIN {X 0,Y 258.465,Z 213.317,A -85,B 0,C 180,E1 -20475.737,E2 -20475.737} C_VEL
LIN {X 0,Y 253.067,Z 203.934,A -85,B 0,C 180,E1 -20477.399,E2 -20477.399} C_VEL
LIN {X 0,Y 246.22,Z 193.248,A -85,B 0,C 180,E1 -20479.643,E2 -20479.643} C_VEL
LIN {X 0,Y 240.854,Z 185.449,A -85,B 0,C 180,E1 -20481.546,E2 -20481.546} C_VEL
LIN {X 0,Y 235.543,Z 178.13,A -85,B 0,C 180,E1 -20483.582,E2 -20483.582} C_VEL
LIN {X 0,Y 232.306,Z 173.809,A -85,B 0,C 180,E1 -20484.913,E2 -20484.913} C_VEL
LIN {X 0,Y 229.772,Z 170.662,A -85,B 0,C 180,E1 -20486.002,E2 -20486.002} C_VEL
LIN {X 0,Y 228.821,Z 169.266,A -85,B 0,C 180,E1 -20486.437,E2 -20486.437} C_VEL
LIN {X 0,Y 226.327,Z 166.663,A -85,B 0,C 180,E1 -20487.558,E2 -20487.558} C_VEL
LIN {X 0,Y 224.872,Z 164.131,A -85,B 0,C 180,E1 -20488.301,E2 -20488.301} C_VEL
LIN {X 0,Y 222.468,Z 162.283,A -85,B 0,C 180,E1 -20489.441,E2 -20489.441} C_VEL
LIN {X 0,Y 221.168,Z 160.042,A -85,B 0,C 180,E1 -20490.165,E2 -20490.165} C_VEL
LIN {X 0,Y 220.847,Z 158.574,A -85,B 0,C 180,E1 -20490.445,E2 -20490.445} C_VEL
LIN {X 0,Y 220.857,Z 158.59,A -85,B 0,C 180,E1 -20493.544,E2 -20493.544} C_VEL
LIN {X 0,Y 220.855,Z 158.588,A -85,B 0,C 180,E1 -20497.551,E2 -20497.551} C_VEL
LIN {X 0,Y 220.921,Z 158.581,A -85,B 0,C 180,E1 -20502.626,E2 -20502.626} C_VEL
LIN {X 0,Y 220.988,Z 158.573,A -85,B 0,C 180,E1 -20507.137,E2 -20507.137} C_VEL
LIN {X 0,Y 221.196,Z 158.542,A -85,B 0,C 180,E1 -20510.859,E2 -20510.859} C_VEL
LIN {X 0,Y 221.112,Z 158.556,A -85,B 0,C 180,E1 -20514.528,E2 -20514.528} C_VEL
LIN {X 0,Y 221.472,Z 158.522,A -85,B 0,C 180,E1 -20518.181,E2 -20518.181} C_VEL
LIN {X 0,Y 221.508,Z 158.515,A -85,B 0,C 180,E1 -20521.818,E2 -20521.818} C_VEL
LIN {X 0,Y 221.216,Z 158.55,A -85,B 0,C 180,E1 -20527.705,E2 -20527.705} C_VEL
LIN {X 0,Y 220.474,Z 158.637,A -85,B 0,C 180,E1 -20529.222,E2 -20529.222} C_VEL
LIN {X 0,Y 217.529,Z 159.017,A -85,B 0,C 180,E1 -20531.695,E2 -20531.695} C_VEL
LIN {X 0,Y 215.053,Z 159.324,A -85,B 0,C 180,E1 -20533.715,E2 -20533.715} C_VEL
LIN {X 0,Y 213.984,Z 159.453,A -85,B 0,C 180,E1 -20535.287,E2 -20535.287} C_VEL
LIN {X 0,Y 213.892,Z 159.459,A -85,B 0,C 180,E1 -20535.82,E2 -20535.82} C_VEL
LIN {X 0,Y 213.831,Z 159.468,A -85,B 0,C 180,E1 -20539.188,E2 -20539.188} C_VEL
LIN {X 0,Y 213.805,Z 159.47,A -85,B 0,C 180,E1 -20543.232,E2 -20543.232} C_VEL
LIN {X 0,Y 213.817,Z 159.468,A -85,B 0,C 180,E1 -20545.753,E2 -20545.753} C_VEL
LIN {X 0,Y 214.586,Z 161.865,A -85,B 0,C 180,E1 -20546.371,E2 -20546.371} C_VEL
LIN {X 0,Y 216.531,Z 164.232,A -85,B 0,C 180,E1 -20547.549,E2 -20547.549} C_VEL
LIN {X 0,Y 218.366,Z 165.505,A -85,B 0,C 180,E1 -20548.538,E2 -20548.538} C_VEL
LIN {X 0,Y 220.165,Z 168.571,A -85,B 0,C 180,E1 -20549.579,E2 -20549.579} C_VEL
LIN {X 0,Y 222.776,Z 171.055,A -85,B 0,C 180,E1 -20550.886,E2 -20550.886} C_VEL
LIN {X 0,Y 225.113,Z 174.384,A -85,B 0,C 180,E1 -20552.055,E2 -20552.055} C_VEL
LIN {X 0,Y 227.742,Z 177.781,A -85,B 0,C 180,E1 -20553.28,E2 -20553.28} C_VEL
LIN {X 0,Y 232.04,Z 184.35,A -85,B 0,C 180,E1 -20555.199,E2 -20555.199} C_VEL
LIN {X 0,Y 235.215,Z 189.277,A -85,B 0,C 180,E1 -20556.522,E2 -20556.522} C_VEL
LIN {X 0,Y 242.391,Z 201.389,A -85,B 0,C 180,E1 -20559.297,E2 -20559.297} C_VEL
LIN {X 0,Y 249.612,Z 215.105,A -85,B 0,C 180,E1 -20561.85,E2 -20561.85} C_VEL
LIN {X 0,Y 255.949,Z 228.832,A -85,B 0,C 180,E1 -20563.945,E2 -20563.945} C_VEL
LIN {X 0,Y 258.985,Z 236.242,A -85,B 0,C 180,E1 -20564.919,E2 -20564.919} C_VEL
LIN {X 0,Y 253.725,Z 326.156,A -85,B 0,C 180,E1 -20567.263,E2 -20567.263} C_VEL
LIN {X 0,Y 251.78,Z 342.318,A -85,B 0,C 180,E1 -20567.939,E2 -20567.939} C_VEL
LIN {X 0,Y 249.107,Z 357.571,A -85,B 0,C 180,E1 -20568.874,E2 -20568.874} C_VEL
LIN {X 0,Y 246.059,Z 371.31,A -85,B 0,C 180,E1 -20570.01,E2 -20570.01} C_VEL
LIN {X 0,Y 242.553,Z 384.817,A -85,B 0,C 180,E1 -20571.474,E2 -20571.474} C_VEL
LIN {X 0,Y 238.813,Z 397.195,A -85,B 0,C 180,E1 -20573.158,E2 -20573.158} C_VEL
LIN {X 0,Y 234.382,Z 409.833,A -85,B 0,C 180,E1 -20575.269,E2 -20575.269} C_VEL
LIN {X 0,Y 230.074,Z 421.324,A -85,B 0,C 180,E1 -20577.685,E2 -20577.685} C_VEL
LIN {X 0,Y 226.262,Z 431.002,A -85,B 0,C 180,E1 -20580.199,E2 -20580.199} C_VEL
LIN {X 0,Y 222.459,Z 440.518,A -85,B 0,C 180,E1 -20583.244,E2 -20583.244} C_VEL
LIN {X 0,Y 219.028,Z 448.444,A -85,B 0,C 180,E1 -20586.353,E2 -20586.353} C_VEL
LIN {X 0,Y 216.014,Z 455.854,A -85,B 0,C 180,E1 -20590.024,E2 -20590.024} C_VEL
LIN {X 0,Y 213.806,Z 461.74,A -85,B 0,C 180,E1 -20593.775,E2 -20593.775} C_VEL
LIN {X 0,Y 212.622,Z 465.244,A -85,B 0,C 180,E1 -20596.622,E2 -20596.622} C_VEL
LIN {X 0,Y 211.718,Z 468.79,A -85,B 0,C 180,E1 -20600.446,E2 -20600.446} C_VEL
LIN {X 0,Y 211.375,Z 471.127,A -85,B 0,C 180,E1 -20604.275,E2 -20604.275} C_VEL
LIN {X 0,Y 211.428,Z 472.306,A -85,B 0,C 180,E1 -20608.095,E2 -20608.095} C_VEL
LIN {X 0,Y 211.544,Z 472.463,A -85,B 0,C 180,E1 -20610,E2 -20610} C_VEL
LIN {X 0,Y 211.356,Z 471.795,A -85,B 0,C 180,E1 -20614.006,E2 -20614.006} C_VEL
LIN {X 0,Y 211.482,Z 470.072,A -85,B 0,C 180,E1 -20617.639,E2 -20617.639} C_VEL
LIN {X 0,Y 212.089,Z 467.124,A -85,B 0,C 180,E1 -20621.468,E2 -20621.468} C_VEL
LIN {X 0,Y 213.376,Z 462.936,A -85,B 0,C 180,E1 -20625.278,E2 -20625.278} C_VEL
LIN {X 0,Y 215.294,Z 457.395,A -85,B 0,C 180,E1 -20629.053,E2 -20629.053} C_VEL
LIN {X 0,Y 218.147,Z 450.361,A -85,B 0,C 180,E1 -20632.743,E2 -20632.743} C_VEL
LIN {X 0,Y 221.371,Z 442.846,A -85,B 0,C 180,E1 -20635.883,E2 -20635.883} C_VEL
LIN {X 0,Y 225.171,Z 433.382,A -85,B 0,C 180,E1 -20639.082,E2 -20639.082} C_VEL
LIN {X 0,Y 229.374,Z 422.905,A -85,B 0,C 180,E1 -20641.907,E2 -20641.907} C_VEL
LIN {X 0,Y 233.977,Z 410.677,A -85,B 0,C 180,E1 -20644.538,E2 -20644.538} C_VEL
LIN {X 0,Y 238.393,Z 398.215,A -85,B 0,C 180,E1 -20646.654,E2 -20646.654} C_VEL
LIN {X 0,Y 242.416,Z 384.86,A -85,B 0,C 180,E1 -20648.485,E2 -20648.485} C_VEL
LIN {X 0,Y 246.042,Z 370.864,A -85,B 0,C 180,E1 -20649.993,E2 -20649.993} C_VEL
LIN {X 0,Y 249.306,Z 355.8,A -85,B 0,C 180,E1 -20651.22,E2 -20651.22} C_VEL
LIN {X 0,Y 251.932,Z 340.703,A -85,B 0,C 180,E1 -20652.097,E2 -20652.097} C_VEL
LIN {X 0,Y 253.59,Z 326.29,A -85,B 0,C 180,E1 -20652.698,E2 -20652.698} C_VEL
LIN {X 0,Y 258.834,Z 236.068,A -85,B 0,C 180,E1 -20655.058,E2 -20655.058} C_VEL
LIN {X 0,Y 252.801,Z 221.899,A -85,B 0,C 180,E1 -20657.008,E2 -20657.008} C_VEL
LIN {X 0,Y 246.063,Z 208.248,A -85,B 0,C 180,E1 -20659.297,E2 -20659.297} C_VEL
LIN {X 0,Y 239.157,Z 195.852,A -85,B 0,C 180,E1 -20661.827,E2 -20661.827} C_VEL
LIN {X 0,Y 233.09,Z 185.941,A -85,B 0,C 180,E1 -20664.257,E2 -20664.257} C_VEL
LIN {X 0,Y 229.231,Z 180.107,A -85,B 0,C 180,E1 -20665.925,E2 -20665.925} C_VEL
LIN {X 0,Y 226.415,Z 175.954,A -85,B 0,C 180,E1 -20667.221,E2 -20667.221} C_VEL
LIN {X 0,Y 223.006,Z 171.494,A -85,B 0,C 180,E1 -20668.864,E2 -20668.864} C_VEL
LIN {X 0,Y 222.317,Z 170.44,A -85,B 0,C 180,E1 -20669.221,E2 -20669.221} C_VEL
LIN {X 0,Y 219.791,Z 168.054,A -85,B 0,C 180,E1 -20670.489,E2 -20670.489} C_VEL
LIN {X 0,Y 218.273,Z 165.218,A -85,B 0,C 180,E1 -20671.383,E2 -20671.383} C_VEL
LIN {X 0,Y 215.672,Z 163.421,A -85,B 0,C 180,E1 -20672.792,E2 -20672.792} C_VEL
LIN {X 0,Y 214.237,Z 161.061,A -85,B 0,C 180,E1 -20673.713,E2 -20673.713} C_VEL
LIN {X 0,Y 213.82,Z 159.47,A -85,B 0,C 180,E1 -20674.117,E2 -20674.117} C_VEL
LIN {X 0,Y 213.853,Z 159.464,A -85,B 0,C 180,E1 -20676.953,E2 -20676.953} C_VEL
LIN {X 0,Y 213.946,Z 159.453,A -85,B 0,C 180,E1 -20682.804,E2 -20682.804} C_VEL
LIN {X 0,Y 213.949,Z 159.451,A -85,B 0,C 180,E1 -20686.706,E2 -20686.706} C_VEL
LIN {X 0,Y 214.135,Z 159.43,A -85,B 0,C 180,E1 -20690.555,E2 -20690.555} C_VEL
LIN {X 0,Y 214.085,Z 159.44,A -85,B 0,C 180,E1 -20694.348,E2 -20694.348} C_VEL
LIN {X 0,Y 214.441,Z 159.4,A -85,B 0,C 180,E1 -20698.122,E2 -20698.122} C_VEL
LIN {X 0,Y 214.516,Z 159.377,A -85,B 0,C 180,E1 -20700,E2 -20700} C_VEL
LIN {X 0,Y 214.409,Z 159.401,A -85,B 0,C 180,E1 -20701.879,E2 -20701.879} C_VEL
LIN {X 0,Y 214.182,Z 159.426,A -85,B 0,C 180,E1 -20707.542,E2 -20707.542} C_VEL
LIN {X 0,Y 213.991,Z 159.455,A -85,B 0,C 180,E1 -20711.365,E2 -20711.365} C_VEL
LIN {X 0,Y 213.881,Z 159.469,A -85,B 0,C 180,E1 -20715.241,E2 -20715.241} C_VEL
LIN {X 0,Y 213.813,Z 159.478,A -85,B 0,C 180,E1 -20719.19,E2 -20719.19} C_VEL
LIN {X 0,Y 213.804,Z 159.478,A -85,B 0,C 180,E1 -20723.232,E2 -20723.232} C_VEL
LIN {X 0,Y 213.85,Z 159.549,A -85,B 0,C 180,E1 -20726.404,E2 -20726.404} C_VEL
LIN {X 0,Y 214.68,Z 162.052,A -85,B 0,C 180,E1 -20727.033,E2 -20727.033} C_VEL
LIN {X 0,Y 216.629,Z 164.32,A -85,B 0,C 180,E1 -20728.193,E2 -20728.193} C_VEL
LIN {X 0,Y 218.292,Z 165.336,A -85,B 0,C 180,E1 -20729.073,E2 -20729.073} C_VEL
LIN {X 0,Y 220.085,Z 168.5,A -85,B 0,C 180,E1 -20730.112,E2 -20730.112} C_VEL
LIN {X 0,Y 222.653,Z 170.886,A -85,B 0,C 180,E1 -20731.389,E2 -20731.389} C_VEL
LIN {X 0,Y 224.964,Z 174.261,A -85,B 0,C 180,E1 -20732.546,E2 -20732.546} C_VEL
LIN {X 0,Y 226.797,Z 176.208,A -85,B 0,C 180,E1 -20733.381,E2 -20733.381} C_VEL
LIN {X 0,Y 229.696,Z 179.989,A -85,B 0,C 180,E1 -20734.678,E2 -20734.678} C_VEL
LIN {X 0,Y 234.388,Z 186.53,A -85,B 0,C 180,E1 -20736.647,E2 -20736.647} C_VEL
LIN {X 0,Y 239.68,Z 193.965,A -85,B 0,C 180,E1 -20738.68,E2 -20738.68} C_VEL
LIN {X 0,Y 246.972,Z 205.263,A -85,B 0,C 180,E1 -20741.256,E2 -20741.256} C_VEL
LIN {X 0,Y 253.571,Z 216.447,A -85,B 0,C 180,E1 -20743.396,E2 -20743.396} C_VEL
LIN {X 0,Y 259.21,Z 228.763,A -85,B 0,C 180,E1 -20745.183,E2 -20745.183} C_VEL
LIN {X 0,Y 254.172,Z 314.862,A -85,B 0,C 180,E1 -20747.423,E2 -20747.423} C_VEL
LIN {X 0,Y 252.386,Z 330.515,A -85,B 0,C 180,E1 -20748.063,E2 -20748.063} C_VEL
LIN {X 0,Y 249.983,Z 346.119,A -85,B 0,C 180,E1 -20749.049,E2 -20749.049} C_VEL
LIN {X 0,Y 246.898,Z 361.305,A -85,B 0,C 180,E1 -20750.364,E2 -20750.364} C_VEL
LIN {X 0,Y 243.498,Z 375.028,A -85,B 0,C 180,E1 -20751.907,E2 -20751.907} C_VEL
LIN {X 0,Y 239.425,Z 388.477,A -85,B 0,C 180,E1 -20753.79,E2 -20753.79} C_VEL
LIN {X 0,Y 235.237,Z 400.682,A -85,B 0,C 180,E1 -20755.932,E2 -20755.932} C_VEL
LIN {X 0,Y 230.921,Z 411.971,A -85,B 0,C 180,E1 -20758.384,E2 -20758.384} C_VEL
LIN {X 0,Y 227.413,Z 421.137,A -85,B 0,C 180,E1 -20760.873,E2 -20760.873} C_VEL
LIN {X 0,Y 223.459,Z 430.325,A -85,B 0,C 180,E1 -20763.876,E2 -20763.876} C_VEL
LIN {X 0,Y 220.105,Z 437.958,A -85,B 0,C 180,E1 -20766.974,E2 -20766.974} C_VEL
LIN {X 0,Y 217.356,Z 444.286,A -85,B 0,C 180,E1 -20770.153,E2 -20770.153} C_VEL
LIN {X 0,Y 214.985,Z 450.093,A -85,B 0,C 180,E1 -20773.867,E2 -20773.867} C_VEL
LIN {X 0,Y 213.642,Z 453.529,A -85,B 0,C 180,E1 -20776.687,E2 -20776.687} C_VEL
LIN {X 0,Y 212.486,Z 457.002,A -85,B 0,C 180,E1 -20780.481,E2 -20780.481} C_VEL
LIN {X 0,Y 211.74,Z 459.473,A -85,B 0,C 180,E1 -20784.718,E2 -20784.718} C_VEL
LIN {X 0,Y 211.558,Z 460.461,A -85,B 0,C 180,E1 -20788.096,E2 -20788.096} C_VEL
LIN {X 0,Y 211.577,Z 460.615,A -85,B 0,C 180,E1 -20790,E2 -20790} C_VEL
LIN {X 0,Y 211.62,Z 460.054,A -85,B 0,C 180,E1 -20793.809,E2 -20793.809} C_VEL
LIN {X 0,Y 212.058,Z 458.379,A -85,B 0,C 180,E1 -20797.618,E2 -20797.618} C_VEL
LIN {X 0,Y 212.936,Z 455.55,A -85,B 0,C 180,E1 -20801.422,E2 -20801.422} C_VEL
LIN {X 0,Y 214.4,Z 451.498,A -85,B 0,C 180,E1 -20805.203,E2 -20805.203} C_VEL
LIN {X 0,Y 216.667,Z 446.116,A -85,B 0,C 180,E1 -20808.927,E2 -20808.927} C_VEL
LIN {X 0,Y 219.598,Z 439.255,A -85,B 0,C 180,E1 -20812.585,E2 -20812.585} C_VEL
LIN {X 0,Y 223.366,Z 430.682,A -85,B 0,C 180,E1 -20816.136,E2 -20816.136} C_VEL
LIN {X 0,Y 227.315,Z 421.561,A -85,B 0,C 180,E1 -20819.141,E2 -20819.141} C_VEL
LIN {X 0,Y 230.913,Z 412.437,A -85,B 0,C 180,E1 -20821.618,E2 -20821.618} C_VEL
LIN {X 0,Y 235.13,Z 401.233,A -85,B 0,C 180,E1 -20824.086,E2 -20824.086} C_VEL
LIN {X 0,Y 239.239,Z 389.135,A -85,B 0,C 180,E1 -20826.243,E2 -20826.243} C_VEL
LIN {X 0,Y 243.363,Z 375.841,A -85,B 0,C 180,E1 -20828.118,E2 -20828.118} C_VEL
LIN {X 0,Y 246.857,Z 361.806,A -85,B 0,C 180,E1 -20829.72,E2 -20829.72} C_VEL
LIN {X 0,Y 250.082,Z 346.265,A -85,B 0,C 180,E1 -20831.064,E2 -20831.064} C_VEL
LIN {X 0,Y 252.544,Z 330.721,A -85,B 0,C 180,E1 -20832.039,E2 -20832.039} C_VEL
LIN {X 0,Y 254.295,Z 315.226,A -85,B 0,C 180,E1 -20832.686,E2 -20832.686} C_VEL
LIN {X 0,Y 258.997,Z 234.321,A -85,B 0,C 180,E1 -20834.804,E2 -20834.804} C_VEL
LIN {X 0,Y 259.242,Z 228.641,A -85,B 0,C 180,E1 -20834.968,E2 -20834.968} C_VEL
LIN {X 0,Y 253.725,Z 216.596,A -85,B 0,C 180,E1 -20836.72,E2 -20836.72} C_VEL
LIN {X 0,Y 246.102,Z 203.716,A -85,B 0,C 180,E1 -20839.214,E2 -20839.214} C_VEL
LIN {X 0,Y 238.676,Z 192.439,A -85,B 0,C 180,E1 -20841.877,E2 -20841.877} C_VEL
LIN {X 0,Y 232.292,Z 183.577,A -85,B 0,C 180,E1 -20844.404,E2 -20844.404} C_VEL
LIN {X 0,Y 229.464,Z 179.746,A -85,B 0,C 180,E1 -20845.618,E2 -20845.618} C_VEL
LIN {X 0,Y 226.595,Z 175.86,A -85,B 0,C 180,E1 -20846.922,E2 -20846.922} C_VEL
LIN {X 0,Y 223.55,Z 172.396,A -85,B 0,C 180,E1 -20848.357,E2 -20848.357} C_VEL
LIN {X 0,Y 222.339,Z 170.468,A -85,B 0,C 180,E1 -20848.989,E2 -20848.989} C_VEL
LIN {X 0,Y 219.755,Z 168.009,A -85,B 0,C 180,E1 -20850.296,E2 -20850.296} C_VEL
LIN {X 0,Y 218.16,Z 165.164,A -85,B 0,C 180,E1 -20851.235,E2 -20851.235} C_VEL
LIN {X 0,Y 215.669,Z 163.482,A -85,B 0,C 180,E1 -20852.594,E2 -20852.594} C_VEL
LIN {X 0,Y 214.243,Z 161.149,A -85,B 0,C 180,E1 -20853.517,E2 -20853.517} C_VEL
LIN {X 0,Y 213.788,Z 159.469,A -85,B 0,C 180,E1 -20853.916,E2 -20853.916} C_VEL
LIN {X 0,Y 213.777,Z 159.474,A -85,B 0,C 180,E1 -20858.799,E2 -20858.799} C_VEL
LIN {X 0,Y 213.885,Z 159.458,A -85,B 0,C 180,E1 -20862.799,E2 -20862.799} C_VEL
LIN {X 0,Y 213.926,Z 159.45,A -85,B 0,C 180,E1 -20866.705,E2 -20866.705} C_VEL
LIN {X 0,Y 214.136,Z 159.422,A -85,B 0,C 180,E1 -20870.555,E2 -20870.555} C_VEL
LIN {X 0,Y 214.076,Z 159.434,A -85,B 0,C 180,E1 -20874.348,E2 -20874.348} C_VEL
LIN {X 0,Y 214.408,Z 159.402,A -85,B 0,C 180,E1 -20878.121,E2 -20878.121} C_VEL
LIN {X 0,Y 214.517,Z 159.374,A -85,B 0,C 180,E1 -20880,E2 -20880} C_VEL
LIN {X 0,Y 214.441,Z 159.396,A -85,B 0,C 180,E1 -20881.878,E2 -20881.878} C_VEL
LIN {X 0,Y 214.177,Z 159.429,A -85,B 0,C 180,E1 -20887.666,E2 -20887.666} C_VEL
LIN {X 0,Y 213.999,Z 159.456,A -85,B 0,C 180,E1 -20891.364,E2 -20891.364} C_VEL
LIN {X 0,Y 213.892,Z 159.459,A -85,B 0,C 180,E1 -20895.82,E2 -20895.82} C_VEL
LIN {X 0,Y 213.189,Z 159.551,A -85,B 0,C 180,E1 -20896.865,E2 -20896.865} C_VEL
LIN {X 0,Y 210.301,Z 159.913,A -85,B 0,C 180,E1 -20898.506,E2 -20898.506} C_VEL
LIN {X 0,Y 207.415,Z 160.278,A -85,B 0,C 180,E1 -20900.19,E2 -20900.19} C_VEL
LIN {X 0,Y 206.758,Z 160.35,A -85,B 0,C 180,E1 -20901.284,E2 -20901.284} C_VEL
LIN {X 0,Y 206.763,Z 160.368,A -85,B 0,C 180,E1 -20901.497,E2 -20901.497} C_VEL
LIN {X 0,Y 207.379,Z 162.534,A -85,B 0,C 180,E1 -20902.116,E2 -20902.116} C_VEL
LIN {X 0,Y 209.271,Z 164.952,A -85,B 0,C 180,E1 -20903.551,E2 -20903.551} C_VEL
LIN {X 0,Y 211.592,Z 166.388,A -85,B 0,C 180,E1 -20905.055,E2 -20905.055} C_VEL
LIN {X 0,Y 213.427,Z 169.597,A -85,B 0,C 180,E1 -20906.319,E2 -20906.319} C_VEL
LIN {X 0,Y 216.141,Z 172.078,A -85,B 0,C 180,E1 -20907.899,E2 -20907.899} C_VEL
LIN {X 0,Y 218.46,Z 175.484,A -85,B 0,C 180,E1 -20909.243,E2 -20909.243} C_VEL
LIN {X 0,Y 220.426,Z 177.461,A -85,B 0,C 180,E1 -20910.262,E2 -20910.262} C_VEL
LIN {X 0,Y 225.087,Z 183.842,A -85,B 0,C 180,E1 -20912.595,E2 -20912.595} C_VEL
LIN {X 0,Y 229.009,Z 189.915,A -85,B 0,C 180,E1 -20914.419,E2 -20914.419} C_VEL
LIN {X 0,Y 232.129,Z 194.97,A -85,B 0,C 180,E1 -20915.782,E2 -20915.782} C_VEL
LIN {X 0,Y 238.716,Z 206.307,A -85,B 0,C 180,E1 -20918.446,E2 -20918.446} C_VEL
LIN {X 0,Y 245.766,Z 219.996,A -85,B 0,C 180,E1 -20921.058,E2 -20921.058} C_VEL
LIN {X 0,Y 252.212,Z 234.418,A -85,B 0,C 180,E1 -20923.29,E2 -20923.29} C_VEL
LIN {X 0,Y 253.856,Z 238.493,A -85,B 0,C 180,E1 -20923.843,E2 -20923.843} C_VEL
LIN {X 0,Y 248.562,Z 325.974,A -85,B 0,C 180,E1 -20926.153,E2 -20926.153} C_VEL
LIN {X 0,Y 246.548,Z 342.128,A -85,B 0,C 180,E1 -20926.832,E2 -20926.832} C_VEL
LIN {X 0,Y 243.811,Z 357.38,A -85,B 0,C 180,E1 -20927.778,E2 -20927.778} C_VEL
LIN {X 0,Y 240.656,Z 371.117,A -85,B 0,C 180,E1 -20928.922,E2 -20928.922} C_VEL
LIN {X 0,Y 236.723,Z 385.642,A -85,B 0,C 180,E1 -20930.525,E2 -20930.525} C_VEL
LIN {X 0,Y 232.725,Z 398.293,A -85,B 0,C 180,E1 -20932.3,E2 -20932.3} C_VEL
LIN {X 0,Y 228.176,Z 410.71,A -85,B 0,C 180,E1 -20934.453,E2 -20934.453} C_VEL
LIN {X 0,Y 223.35,Z 422.89,A -85,B 0,C 180,E1 -20937.126,E2 -20937.126} C_VEL
LIN {X 0,Y 218.87,Z 433.627,A -85,B 0,C 180,E1 -20940.109,E2 -20940.109} C_VEL
LIN {X 0,Y 215.008,Z 442.775,A -85,B 0,C 180,E1 -20943.291,E2 -20943.291} C_VEL
LIN {X 0,Y 211.548,Z 450.275,A -85,B 0,C 180,E1 -20946.505,E2 -20946.505} C_VEL
LIN {X 0,Y 208.634,Z 457.282,A -85,B 0,C 180,E1 -20950.314,E2 -20950.314} C_VEL
LIN {X 0,Y 206.484,Z 462.797,A -85,B 0,C 180,E1 -20954.199,E2 -20954.199} C_VEL
LIN {X 0,Y 205.068,Z 466.972,A -85,B 0,C 180,E1 -20958.134,E2 -20958.134} C_VEL
LIN {X 0,Y 204.414,Z 469.907,A -85,B 0,C 180,E1 -20962.095,E2 -20962.095} C_VEL
LIN {X 0,Y 204.259,Z 471.698,A -85,B 0,C 180,E1 -20966.207,E2 -20966.207} C_VEL
LIN {X 0,Y 204.461,Z 472.265,A -85,B 0,C 180,E1 -20970,E2 -20970} C_VEL
LIN {X 0,Y 204.259,Z 471.646,A -85,B 0,C 180,E1 -20973.946,E2 -20973.946} C_VEL
LIN {X 0,Y 204.414,Z 469.872,A -85,B 0,C 180,E1 -20977.905,E2 -20977.905} C_VEL
LIN {X 0,Y 205.066,Z 466.923,A -85,B 0,C 180,E1 -20981.866,E2 -20981.866} C_VEL
LIN {X 0,Y 206.445,Z 462.734,A -85,B 0,C 180,E1 -20985.804,E2 -20985.804} C_VEL
LIN {X 0,Y 208.544,Z 457.194,A -85,B 0,C 180,E1 -20989.694,E2 -20989.694} C_VEL
LIN {X 0,Y 211.532,Z 450.158,A -85,B 0,C 180,E1 -20993.496,E2 -20993.496} C_VEL
LIN {X 0,Y 214.959,Z 442.644,A -85,B 0,C 180,E1 -20996.715,E2 -20996.715} C_VEL
LIN {X 0,Y 218.664,Z 433.795,A -85,B 0,C 180,E1 -20999.797,E2 -20999.797} C_VEL
LIN {X 0,Y 223.337,Z 422.703,A -85,B 0,C 180,E1 -21002.876,E2 -21002.876} C_VEL
LIN {X 0,Y 228.114,Z 410.473,A -85,B 0,C 180,E1 -21005.558,E2 -21005.558} C_VEL
LIN {X 0,Y 232.7,Z 398.011,A -85,B 0,C 180,E1 -21007.705,E2 -21007.705} C_VEL
LIN {X 0,Y 236.906,Z 384.564,A -85,B 0,C 180,E1 -21009.569,E2 -21009.569} C_VEL
LIN {X 0,Y 240.654,Z 370.659,A -85,B 0,C 180,E1 -21011.078,E2 -21011.078} C_VEL
LIN {X 0,Y 244.02,Z 355.594,A -85,B 0,C 180,E1 -21012.316,E2 -21012.316} C_VEL
LIN {X 0,Y 246.698,Z 340.493,A -85,B 0,C 180,E1 -21013.205,E2 -21013.205} C_VEL
LIN {X 0,Y 248.533,Z 324.603,A -85,B 0,C 180,E1 -21013.853,E2 -21013.853} C_VEL
LIN {X 0,Y 253.741,Z 238.52,A -85,B 0,C 180,E1 -21016.116,E2 -21016.116} C_VEL
LIN {X 0,Y 248.307,Z 225.586,A -85,B 0,C 180,E1 -21017.967,E2 -21017.967} C_VEL
LIN {X 0,Y 242.249,Z 213.104,A -85,B 0,C 180,E1 -21020.129,E2 -21020.129} C_VEL
LIN {X 0,Y 235.766,Z 201.185,A -85,B 0,C 180,E1 -21022.618,E2 -21022.618} C_VEL
LIN {X 0,Y 230.202,Z 191.834,A -85,B 0,C 180,E1 -21024.947,E2 -21024.947} C_VEL
LIN {X 0,Y 226.662,Z 186.322,A -85,B 0,C 180,E1 -21026.54,E2 -21026.54} C_VEL
LIN {X 0,Y 223.252,Z 181.233,A -85,B 0,C 180,E1 -21028.178,E2 -21028.178} C_VEL
LIN {X 0,Y 220.251,Z 177.185,A -85,B 0,C 180,E1 -21029.701,E2 -21029.701} C_VEL
LIN {X 0,Y 217.047,Z 173.647,A -85,B 0,C 180,E1 -21031.405,E2 -21031.405} C_VEL
LIN {X 0,Y 215.802,Z 171.619,A -85,B 0,C 180,E1 -21032.152,E2 -21032.152} C_VEL
LIN {X 0,Y 213.225,Z 169.337,A -85,B 0,C 180,E1 -21033.647,E2 -21033.647} C_VEL
LIN {X 0,Y 211.372,Z 166.149,A -85,B 0,C 180,E1 -21034.917,E2 -21034.917} C_VEL
LIN {X 0,Y 208.792,Z 164.463,A -85,B 0,C 180,E1 -21036.6,E2 -21036.6} C_VEL
LIN {X 0,Y 207.186,Z 161.999,A -85,B 0,C 180,E1 -21037.856,E2 -21037.856} C_VEL
LIN {X 0,Y 206.766,Z 160.356,A -85,B 0,C 180,E1 -21038.307,E2 -21038.307} C_VEL
LIN {X 0,Y 206.875,Z 160.339,A -85,B 0,C 180,E1 -21042.197,E2 -21042.197} C_VEL
LIN {X 0,Y 206.892,Z 160.334,A -85,B 0,C 180,E1 -21046.244,E2 -21046.244} C_VEL
LIN {X 0,Y 207.08,Z 160.311,A -85,B 0,C 180,E1 -21050.23,E2 -21050.23} C_VEL
LIN {X 0,Y 207.047,Z 160.319,A -85,B 0,C 180,E1 -21054.156,E2 -21054.156} C_VEL
LIN {X 0,Y 207.377,Z 160.279,A -85,B 0,C 180,E1 -21058.058,E2 -21058.058} C_VEL
LIN {X 0,Y 207.484,Z 160.253,A -85,B 0,C 180,E1 -21060,E2 -21060} C_VEL
LIN {X 0,Y 207.348,Z 160.28,A -85,B 0,C 180,E1 -21061.943,E2 -21061.943} C_VEL
LIN {X 0,Y 207.127,Z 160.302,A -85,B 0,C 180,E1 -21067.801,E2 -21067.801} C_VEL
LIN {X 0,Y 206.911,Z 160.332,A -85,B 0,C 180,E1 -21071.759,E2 -21071.759} C_VEL
LIN {X 0,Y 206.815,Z 160.345,A -85,B 0,C 180,E1 -21075.775,E2 -21075.775} C_VEL
LIN {X 0,Y 206.748,Z 160.352,A -85,B 0,C 180,E1 -21079.873,E2 -21079.873} C_VEL
LIN {X 0,Y 206.75,Z 160.472,A -85,B 0,C 180,E1 -21082.149,E2 -21082.149} C_VEL
LIN {X 0,Y 207.51,Z 162.744,A -85,B 0,C 180,E1 -21082.865,E2 -21082.865} C_VEL
LIN {X 0,Y 209.249,Z 164.946,A -85,B 0,C 180,E1 -21084.164,E2 -21084.164} C_VEL
LIN {X 0,Y 211.571,Z 166.279,A -85,B 0,C 180,E1 -21085.646,E2 -21085.646} C_VEL
LIN {X 0,Y 213.277,Z 169.452,A -85,B 0,C 180,E1 -21086.828,E2 -21086.828} C_VEL
LIN {X 0,Y 216.103,Z 172.054,A -85,B 0,C 180,E1 -21088.467,E2 -21088.467} C_VEL
LIN {X 0,Y 218.38,Z 175.419,A -85,B 0,C 180,E1 -21089.779,E2 -21089.779} C_VEL
LIN {X 0,Y 220.383,Z 177.453,A -85,B 0,C 180,E1 -21090.813,E2 -21090.813} C_VEL
LIN {X 0,Y 223.176,Z 181.143,A -85,B 0,C 180,E1 -21092.225,E2 -21092.225} C_VEL
LIN {X 0,Y 224.746,Z 183.18,A -85,B 0,C 180,E1 -21092.978,E2 -21092.978} C_VEL
LIN {X 0,Y 228.095,Z 187.673,A -85,B 0,C 180,E1 -21094.51,E2 -21094.51} C_VEL
LIN {X 0,Y 233.534,Z 195.208,A -85,B 0,C 180,E1 -21096.803,E2 -21096.803} C_VEL
LIN {X 0,Y 241.081,Z 206.699,A -85,B 0,C 180,E1 -21099.686,E2 -21099.686} C_VEL
LIN {X 0,Y 248.633,Z 219.486,A -85,B 0,C 180,E1 -21102.297,E2 -21102.297} C_VEL
LIN {X 0,Y 252.662,Z 227.853,A -85,B 0,C 180,E1 -21103.64,E2 -21103.64} C_VEL
LIN {X 0,Y 254.117,Z 231.187,A -85,B 0,C 180,E1 -21104.119,E2 -21104.119} C_VEL
LIN {X 0,Y 249.008,Z 315.08,A -85,B 0,C 180,E1 -21106.322,E2 -21106.322} C_VEL
LIN {X 0,Y 247.155,Z 330.725,A -85,B 0,C 180,E1 -21106.964,E2 -21106.964} C_VEL
LIN {X 0,Y 244.662,Z 346.326,A -85,B 0,C 180,E1 -21107.959,E2 -21107.959} C_VEL
LIN {X 0,Y 241.477,Z 361.51,A -85,B 0,C 180,E1 -21109.29,E2 -21109.29} C_VEL
LIN {X 0,Y 237.946,Z 375.232,A -85,B 0,C 180,E1 -21110.851,E2 -21110.851} C_VEL
LIN {X 0,Y 233.72,Z 388.68,A -85,B 0,C 180,E1 -21112.759,E2 -21112.759} C_VEL
LIN {X 0,Y 229.387,Z 400.884,A -85,B 0,C 180,E1 -21114.938,E2 -21114.938} C_VEL
LIN {X 0,Y 224.884,Z 412.173,A -85,B 0,C 180,E1 -21117.432,E2 -21117.432} C_VEL
LIN {X 0,Y 221.224,Z 421.339,A -85,B 0,C 180,E1 -21119.976,E2 -21119.976} C_VEL
LIN {X 0,Y 217.088,Z 430.527,A -85,B 0,C 180,E1 -21123.049,E2 -21123.049} C_VEL
LIN {X 0,Y 213.563,Z 438.159,A -85,B 0,C 180,E1 -21126.226,E2 -21126.226} C_VEL
LIN {X 0,Y 210.633,Z 444.537,A -85,B 0,C 180,E1 -21129.523,E2 -21129.523} C_VEL
LIN {X 0,Y 208.15,Z 450.293,A -85,B 0,C 180,E1 -21133.322,E2 -21133.322} C_VEL
LIN {X 0,Y 206.718,Z 453.729,A -85,B 0,C 180,E1 -21136.232,E2 -21136.232} C_VEL
LIN {X 0,Y 205.464,Z 457.202,A -85,B 0,C 180,E1 -21140.152,E2 -21140.152} C_VEL
LIN {X 0,Y 204.71,Z 459.495,A -85,B 0,C 180,E1 -21144.088,E2 -21144.088} C_VEL
LIN {X 0,Y 204.462,Z 460.66,A -85,B 0,C 180,E1 -21148.03,E2 -21148.03} C_VEL
LIN {X 0,Y 204.496,Z 460.814,A -85,B 0,C 180,E1 -21150,E2 -21150} C_VEL
LIN {X 0,Y 204.54,Z 460.252,A -85,B 0,C 180,E1 -21153.941,E2 -21153.941} C_VEL
LIN {X 0,Y 205.009,Z 458.577,A -85,B 0,C 180,E1 -21157.882,E2 -21157.882} C_VEL
LIN {X 0,Y 205.942,Z 455.749,A -85,B 0,C 180,E1 -21161.815,E2 -21161.815} C_VEL
LIN {X 0,Y 207.524,Z 451.696,A -85,B 0,C 180,E1 -21165.72,E2 -21165.72} C_VEL
LIN {X 0,Y 209.912,Z 446.315,A -85,B 0,C 180,E1 -21169.561,E2 -21169.561} C_VEL
LIN {X 0,Y 213.014,Z 439.453,A -85,B 0,C 180,E1 -21173.323,E2 -21173.323} C_VEL
LIN {X 0,Y 217.007,Z 430.879,A -85,B 0,C 180,E1 -21176.963,E2 -21176.963} C_VEL
LIN {X 0,Y 221.124,Z 421.758,A -85,B 0,C 180,E1 -21180.039,E2 -21180.039} C_VEL
LIN {X 0,Y 224.869,Z 412.634,A -85,B 0,C 180,E1 -21182.571,E2 -21182.571} C_VEL
LIN {X 0,Y 229.282,Z 401.428,A -85,B 0,C 180,E1 -21185.081,E2 -21185.081} C_VEL
LIN {X 0,Y 233.538,Z 389.33,A -85,B 0,C 180,E1 -21187.275,E2 -21187.275} C_VEL
LIN {X 0,Y 237.814,Z 376.035,A -85,B 0,C 180,E1 -21189.175,E2 -21189.175} C_VEL
LIN {X 0,Y 241.279,Z 362.606,A -85,B 0,C 180,E1 -21190.734,E2 -21190.734} C_VEL
LIN {X 0,Y 244.546,Z 347.607,A -85,B 0,C 180,E1 -21192.066,E2 -21192.066} C_VEL
LIN {X 0,Y 247.206,Z 331.762,A -85,B 0,C 180,E1 -21193.095,E2 -21193.095} C_VEL
LIN {X 0,Y 248.985,Z 316.709,A -85,B 0,C 180,E1 -21193.753,E2 -21193.753} C_VEL
LIN {X 0,Y 253.632,Z 241.543,A -85,B 0,C 180,E1 -21195.739,E2 -21195.739} C_VEL
LIN {X 0,Y 254.106,Z 231.001,A -85,B 0,C 180,E1 -21196.049,E2 -21196.049} C_VEL
LIN {X 0,Y 249.125,Z 220.215,A -85,B 0,C 180,E1 -21197.71,E2 -21197.71} C_VEL
LIN {X 0,Y 241.768,Z 207.721,A -85,B 0,C 180,E1 -21200.244,E2 -21200.244} C_VEL
LIN {X 0,Y 234.946,Z 197.295,A -85,B 0,C 180,E1 -21202.817,E2 -21202.817} C_VEL
LIN {X 0,Y 229.254,Z 189.195,A -85,B 0,C 180,E1 -21205.182,E2 -21205.182} C_VEL
LIN {X 0,Y 226.258,Z 185.143,A -85,B 0,C 180,E1 -21206.525,E2 -21206.525} C_VEL
LIN {X 0,Y 223.214,Z 181.136,A -85,B 0,C 180,E1 -21207.972,E2 -21207.972} C_VEL
LIN {X 0,Y 220.514,Z 177.613,A -85,B 0,C 180,E1 -21209.34,E2 -21209.34} C_VEL
LIN {X 0,Y 219.632,Z 176.543,A -85,B 0,C 180,E1 -21209.802,E2 -21209.802} C_VEL
LIN {X 0,Y 216.948,Z 173.498,A -85,B 0,C 180,E1 -21211.258,E2 -21211.258} C_VEL
LIN {X 0,Y 215.799,Z 171.637,A -85,B 0,C 180,E1 -21211.953,E2 -21211.953} C_VEL
LIN {X 0,Y 213.12,Z 169.26,A -85,B 0,C 180,E1 -21213.524,E2 -21213.524} C_VEL
LIN {X 0,Y 211.491,Z 166.205,A -85,B 0,C 180,E1 -21214.669,E2 -21214.669} C_VEL
LIN {X 0,Y 208.829,Z 164.581,A -85,B 0,C 180,E1 -21216.409,E2 -21216.409} C_VEL
LIN {X 0,Y 207.177,Z 162.08,A -85,B 0,C 180,E1 -21217.712,E2 -21217.712} C_VEL
LIN {X 0,Y 206.728,Z 160.348,A -85,B 0,C 180,E1 -21218.236,E2 -21218.236} C_VEL
LIN {X 0,Y 206.805,Z 160.337,A -85,B 0,C 180,E1 -21222.19,E2 -21222.19} C_VEL
LIN {X 0,Y 206.866,Z 160.328,A -85,B 0,C 180,E1 -21226.242,E2 -21226.242} C_VEL
LIN {X 0,Y 207.08,Z 160.301,A -85,B 0,C 180,E1 -21230.23,E2 -21230.23} C_VEL
LIN {X 0,Y 207.039,Z 160.312,A -85,B 0,C 180,E1 -21234.155,E2 -21234.155} C_VEL
LIN {X 0,Y 207.347,Z 160.282,A -85,B 0,C 180,E1 -21238.057,E2 -21238.057} C_VEL
LIN {X 0,Y 207.484,Z 160.25,A -85,B 0,C 180,E1 -21240,E2 -21240} C_VEL
LIN {X 0,Y 207.377,Z 160.276,A -85,B 0,C 180,E1 -21241.942,E2 -21241.942} C_VEL
LIN {X 0,Y 207.132,Z 160.305,A -85,B 0,C 180,E1 -21247.8,E2 -21247.8} C_VEL
LIN {X 0,Y 206.923,Z 160.338,A -85,B 0,C 180,E1 -21251.758,E2 -21251.758} C_VEL
LIN {X 0,Y 206.848,Z 160.347,A -85,B 0,C 180,E1 -21255.793,E2 -21255.793} C_VEL
LIN {X 0,Y 206.777,Z 160.353,A -85,B 0,C 180,E1 -21259.87,E2 -21259.87} C_VEL
LIN {X 0,Y 206.758,Z 160.35,A -85,B 0,C 180,E1 -21261.284,E2 -21261.284} C_VEL
LIN {X 0,Y 207.759,Z 161.053,A -85,B 0,C 180,E1 -21262.24,E2 -21262.24} C_VEL
LIN {X 0,Y 209.152,Z 163.336,A -85,B 0,C 180,E1 -21263.321,E2 -21263.321} C_VEL
LIN {X 0,Y 210.672,Z 167.967,A -85,B 0,C 180,E1 -21264.644,E2 -21264.644} C_VEL
LIN {X 0,Y 212.506,Z 174.288,A -85,B 0,C 180,E1 -21266.078,E2 -21266.078} C_VEL
LIN {X 0,Y 213.991,Z 178.532,A -85,B 0,C 180,E1 -21267.255,E2 -21267.255} C_VEL
LIN {X 0,Y 214.648,Z 179.705,A -85,B 0,C 180,E1 -21267.683,E2 -21267.683} C_VEL
LIN {X 0,Y 217.643,Z 183.119,A -85,B 0,C 180,E1 -21269.364,E2 -21269.364} C_VEL
LIN {X 0,Y 222.153,Z 189.355,A -85,B 0,C 180,E1 -21271.732,E2 -21271.732} C_VEL
LIN {X 0,Y 228.168,Z 198.975,A -85,B 0,C 180,E1 -21274.604,E2 -21274.604} C_VEL
LIN {X 0,Y 235.34,Z 211.681,A -85,B 0,C 180,E1 -21277.668,E2 -21277.668} C_VEL
LIN {X 0,Y 242.361,Z 225.683,A -85,B 0,C 180,E1 -21280.385,E2 -21280.385} C_VEL
LIN {X 0,Y 248.619,Z 240.255,A -85,B 0,C 180,E1 -21282.653,E2 -21282.653} C_VEL
LIN {X 0,Y 248.86,Z 241.279,A -85,B 0,C 180,E1 -21282.755,E2 -21282.755} C_VEL
LIN {X 0,Y 243.495,Z 325.792,A -85,B 0,C 180,E1 -21284.997,E2 -21284.997} C_VEL
LIN {X 0,Y 241.418,Z 341.938,A -85,B 0,C 180,E1 -21285.679,E2 -21285.679} C_VEL
LIN {X 0,Y 238.608,Z 357.188,A -85,B 0,C 180,E1 -21286.634,E2 -21286.634} C_VEL
LIN {X 0,Y 235.336,Z 370.923,A -85,B 0,C 180,E1 -21287.783,E2 -21287.783} C_VEL
LIN {X 0,Y 231.566,Z 384.452,A -85,B 0,C 180,E1 -21289.28,E2 -21289.28} C_VEL
LIN {X 0,Y 227.112,Z 398.097,A -85,B 0,C 180,E1 -21291.197,E2 -21291.197} C_VEL
LIN {X 0,Y 222.391,Z 410.513,A -85,B 0,C 180,E1 -21293.381,E2 -21293.381} C_VEL
LIN {X 0,Y 217.382,Z 422.693,A -85,B 0,C 180,E1 -21296.103,E2 -21296.103} C_VEL
LIN {X 0,Y 212.836,Z 433.163,A -85,B 0,C 180,E1 -21299.064,E2 -21299.064} C_VEL
LIN {X 0,Y 208.63,Z 442.576,A -85,B 0,C 180,E1 -21302.407,E2 -21302.407} C_VEL
LIN {X 0,Y 205.007,Z 450.076,A -85,B 0,C 180,E1 -21305.708,E2 -21305.708} C_VEL
LIN {X 0,Y 201.874,Z 457.082,A -85,B 0,C 180,E1 -21309.626,E2 -21309.626} C_VEL
LIN {X 0,Y 199.58,Z 462.597,A -85,B 0,C 180,E1 -21313.637,E2 -21313.637} C_VEL
LIN {X 0,Y 198.06,Z 466.772,A -85,B 0,C 180,E1 -21317.707,E2 -21317.707} C_VEL
LIN {X 0,Y 197.339,Z 469.707,A -85,B 0,C 180,E1 -21321.81,E2 -21321.81} C_VEL
LIN {X 0,Y 197.171,Z 471.462,A -85,B 0,C 180,E1 -21325.912,E2 -21325.912} C_VEL
LIN {X 0,Y 197.361,Z 472.066,A -85,B 0,C 180,E1 -21330,E2 -21330} C_VEL
LIN {X 0,Y 197.171,Z 471.446,A -85,B 0,C 180,E1 -21334.088,E2 -21334.088} C_VEL
LIN {X 0,Y 197.339,Z 469.672,A -85,B 0,C 180,E1 -21338.19,E2 -21338.19} C_VEL
LIN {X 0,Y 198.057,Z 466.721,A -85,B 0,C 180,E1 -21342.293,E2 -21342.293} C_VEL
LIN {X 0,Y 199.539,Z 462.532,A -85,B 0,C 180,E1 -21346.366,E2 -21346.366} C_VEL
LIN {X 0,Y 201.808,Z 456.992,A -85,B 0,C 180,E1 -21350.38,E2 -21350.38} C_VEL
LIN {X 0,Y 204.989,Z 449.956,A -85,B 0,C 180,E1 -21354.294,E2 -21354.294} C_VEL
LIN {X 0,Y 208.575,Z 442.442,A -85,B 0,C 180,E1 -21357.601,E2 -21357.601} C_VEL
LIN {X 0,Y 212.659,Z 433.218,A -85,B 0,C 180,E1 -21360.879,E2 -21360.879} C_VEL
LIN {X 0,Y 217.371,Z 422.5,A -85,B 0,C 180,E1 -21363.899,E2 -21363.899} C_VEL
LIN {X 0,Y 222.363,Z 410.27,A -85,B 0,C 180,E1 -21366.624,E2 -21366.624} C_VEL
LIN {X 0,Y 227.105,Z 397.807,A -85,B 0,C 180,E1 -21368.804,E2 -21368.804} C_VEL
LIN {X 0,Y 231.255,Z 385.036,A -85,B 0,C 180,E1 -21370.611,E2 -21370.611} C_VEL
LIN {X 0,Y 235.342,Z 370.454,A -85,B 0,C 180,E1 -21372.215,E2 -21372.215} C_VEL
LIN {X 0,Y 238.812,Z 355.387,A -85,B 0,C 180,E1 -21373.465,E2 -21373.465} C_VEL
LIN {X 0,Y 241.568,Z 340.283,A -85,B 0,C 180,E1 -21374.359,E2 -21374.359} C_VEL
LIN {X 0,Y 243.457,Z 324.385,A -85,B 0,C 180,E1 -21375.012,E2 -21375.012} C_VEL
LIN {X 0,Y 248.729,Z 240.771,A -85,B 0,C 180,E1 -21377.227,E2 -21377.227} C_VEL
LIN {X 0,Y 243.186,Z 227.796,A -85,B 0,C 180,E1 -21379.215,E2 -21379.215} C_VEL
LIN {X 0,Y 237.267,Z 215.479,A -85,B 0,C 180,E1 -21381.468,E2 -21381.468} C_VEL
LIN {X 0,Y 230.053,Z 202.24,A -85,B 0,C 180,E1 -21384.451,E2 -21384.451} C_VEL
LIN {X 0,Y 225.549,Z 194.812,A -85,B 0,C 180,E1 -21386.487,E2 -21386.487} C_VEL
LIN {X 0,Y 220.664,Z 187.22,A -85,B 0,C 180,E1 -21388.899,E2 -21388.899} C_VEL
LIN {X 0,Y 217.245,Z 182.752,A -85,B 0,C 180,E1 -21390.706,E2 -21390.706} C_VEL
LIN {X 0,Y 214.497,Z 179.444,A -85,B 0,C 180,E1 -21392.26,E2 -21392.26} C_VEL
LIN {X 0,Y 213.5,Z 177.961,A -85,B 0,C 180,E1 -21392.875,E2 -21392.875} C_VEL
LIN {X 0,Y 210.918,Z 175.353,A -85,B 0,C 180,E1 -21394.463,E2 -21394.463} C_VEL
LIN {X 0,Y 209.51,Z 172.851,A -85,B 0,C 180,E1 -21395.473,E2 -21395.473} C_VEL
LIN {X 0,Y 206.887,Z 170.866,A -85,B 0,C 180,E1 -21397.272,E2 -21397.272} C_VEL
LIN {X 0,Y 205.133,Z 168.067,A -85,B 0,C 180,E1 -21398.719,E2 -21398.719} C_VEL
LIN {X 0,Y 204.681,Z 167.137,A -85,B 0,C 180,E1 -21399.131,E2 -21399.131} C_VEL
LIN {X 0,Y 201.959,Z 165.526,A -85,B 0,C 180,E1 -21401.407,E2 -21401.407} C_VEL
LIN {X 0,Y 200.281,Z 162.992,A -85,B 0,C 180,E1 -21403.172,E2 -21403.172} C_VEL
LIN {X 0,Y 199.829,Z 161.208,A -85,B 0,C 180,E1 -21403.921,E2 -21403.921} C_VEL
LIN {X 0,Y 200.024,Z 161.194,A -85,B 0,C 180,E1 -21409.882,E2 -21409.882} C_VEL
LIN {X 0,Y 200.009,Z 161.197,A -85,B 0,C 180,E1 -21413.949,E2 -21413.949} C_VEL
LIN {X 0,Y 200.316,Z 161.159,A -85,B 0,C 180,E1 -21417.99,E2 -21417.99} C_VEL
LIN {X 0,Y 200.451,Z 161.128,A -85,B 0,C 180,E1 -21420,E2 -21420} C_VEL
LIN {X 0,Y 199.993,Z 161.186,A -85,B 0,C 180,E1 -21424.03,E2 -21424.03} C_VEL
LIN {X 0,Y 200.075,Z 161.178,A -85,B 0,C 180,E1 -21428.077,E2 -21428.077} C_VEL
LIN {X 0,Y 199.86,Z 161.206,A -85,B 0,C 180,E1 -21432.18,E2 -21432.18} C_VEL
LIN {X 0,Y 199.75,Z 161.246,A -85,B 0,C 180,E1 -21436.545,E2 -21436.545} C_VEL
LIN {X 0,Y 200.388,Z 163.377,A -85,B 0,C 180,E1 -21437.412,E2 -21437.412} C_VEL
LIN {X 0,Y 202.22,Z 165.818,A -85,B 0,C 180,E1 -21439.279,E2 -21439.279} C_VEL
LIN {X 0,Y 204.839,Z 167.385,A -85,B 0,C 180,E1 -21441.446,E2 -21441.446} C_VEL
LIN {X 0,Y 206.36,Z 170.302,A -85,B 0,C 180,E1 -21442.769,E2 -21442.769} C_VEL
LIN {X 0,Y 208.602,Z 172.337,A -85,B 0,C 180,E1 -21444.376,E2 -21444.376} C_VEL
LIN {X 0,Y 209.636,Z 173.143,A -85,B 0,C 180,E1 -21445.064,E2 -21445.064} C_VEL
LIN {X 0,Y 211.7,Z 176.381,A -85,B 0,C 180,E1 -21446.488,E2 -21446.488} C_VEL
LIN {X 0,Y 213.959,Z 178.553,A -85,B 0,C 180,E1 -21447.843,E2 -21447.843} C_VEL
LIN {X 0,Y 216.501,Z 182.083,A -85,B 0,C 180,E1 -21449.339,E2 -21449.339} C_VEL
LIN {X 0,Y 218.051,Z 183.799,A -85,B 0,C 180,E1 -21450.173,E2 -21450.173} C_VEL
LIN {X 0,Y 222.223,Z 189.358,A -85,B 0,C 180,E1 -21452.322,E2 -21452.322} C_VEL
LIN {X 0,Y 225.677,Z 194.074,A -85,B 0,C 180,E1 -21453.96,E2 -21453.96} C_VEL
LIN {X 0,Y 230.723,Z 201.313,A -85,B 0,C 180,E1 -21456.17,E2 -21456.17} C_VEL
LIN {X 0,Y 237.655,Z 212.049,A -85,B 0,C 180,E1 -21458.925,E2 -21458.925} C_VEL
LIN {X 0,Y 245.118,Z 224.961,A -85,B 0,C 180,E1 -21461.617,E2 -21461.617} C_VEL
LIN {X 0,Y 249.094,Z 233.627,A -85,B 0,C 180,E1 -21463.006,E2 -21463.006} C_VEL
LIN {X 0,Y 243.939,Z 315.298,A -85,B 0,C 180,E1 -21465.174,E2 -21465.174} C_VEL
LIN {X 0,Y 242.025,Z 330.936,A -85,B 0,C 180,E1 -21465.819,E2 -21465.819} C_VEL
LIN {X 0,Y 239.453,Z 346.533,A -85,B 0,C 180,E1 -21466.825,E2 -21466.825} C_VEL
LIN {X 0,Y 236.23,Z 361.334,A -85,B 0,C 180,E1 -21468.126,E2 -21468.126} C_VEL
LIN {X 0,Y 232.492,Z 375.435,A -85,B 0,C 180,E1 -21469.748,E2 -21469.748} C_VEL
LIN {X 0,Y 228.093,Z 388.884,A -85,B 0,C 180,E1 -21471.677,E2 -21471.677} C_VEL
LIN {X 0,Y 223.616,Z 401.086,A -85,B 0,C 180,E1 -21473.893,E2 -21473.893} C_VEL
LIN {X 0,Y 218.989,Z 412.205,A -85,B 0,C 180,E1 -21476.385,E2 -21476.385} C_VEL
LIN {X 0,Y 214.417,Z 422.987,A -85,B 0,C 180,E1 -21479.466,E2 -21479.466} C_VEL
LIN {X 0,Y 210.186,Z 431.944,A -85,B 0,C 180,E1 -21482.628,E2 -21482.628} C_VEL
LIN {X 0,Y 206.555,Z 439.361,A -85,B 0,C 180,E1 -21485.902,E2 -21485.902} C_VEL
LIN {X 0,Y 203.239,Z 446.287,A -85,B 0,C 180,E1 -21489.769,E2 -21489.769} C_VEL
LIN {X 0,Y 200.71,Z 451.723,A -85,B 0,C 180,E1 -21493.732,E2 -21493.732} C_VEL
LIN {X 0,Y 199.031,Z 455.818,A -85,B 0,C 180,E1 -21497.768,E2 -21497.768} C_VEL
LIN {X 0,Y 197.966,Z 458.692,A -85,B 0,C 180,E1 -21501.836,E2 -21501.836} C_VEL
LIN {X 0,Y 197.463,Z 460.415,A -85,B 0,C 180,E1 -21505.918,E2 -21505.918} C_VEL
LIN {X 0,Y 197.397,Z 461.012,A -85,B 0,C 180,E1 -21510,E2 -21510} C_VEL
LIN {X 0,Y 197.463,Z 460.451,A -85,B 0,C 180,E1 -21514.082,E2 -21514.082} C_VEL
LIN {X 0,Y 197.956,Z 458.776,A -85,B 0,C 180,E1 -21518.164,E2 -21518.164} C_VEL
LIN {X 0,Y 198.97,Z 455.948,A -85,B 0,C 180,E1 -21522.236,E2 -21522.236} C_VEL
LIN {X 0,Y 200.672,Z 451.895,A -85,B 0,C 180,E1 -21526.271,E2 -21526.271} C_VEL
LIN {X 0,Y 203.192,Z 446.513,A -85,B 0,C 180,E1 -21530.236,E2 -21530.236} C_VEL
LIN {X 0,Y 206.486,Z 439.651,A -85,B 0,C 180,E1 -21534.107,E2 -21534.107} C_VEL
LIN {X 0,Y 210.671,Z 431.077,A -85,B 0,C 180,E1 -21537.843,E2 -21537.843} C_VEL
LIN {X 0,Y 214.328,Z 423.365,A -85,B 0,C 180,E1 -21540.548,E2 -21540.548} C_VEL
LIN {X 0,Y 218.954,Z 412.668,A -85,B 0,C 180,E1 -21543.621,E2 -21543.621} C_VEL
LIN {X 0,Y 223.517,Z 401.623,A -85,B 0,C 180,E1 -21546.125,E2 -21546.125} C_VEL
LIN {X 0,Y 227.933,Z 389.525,A -85,B 0,C 180,E1 -21548.355,E2 -21548.355} C_VEL
LIN {X 0,Y 232.35,Z 376.23,A -85,B 0,C 180,E1 -21550.282,E2 -21550.282} C_VEL
LIN {X 0,Y 235.96,Z 362.692,A -85,B 0,C 180,E1 -21551.874,E2 -21551.874} C_VEL
LIN {X 0,Y 239.34,Z 347.798,A -85,B 0,C 180,E1 -21553.2,E2 -21553.2} C_VEL
LIN {X 0,Y 242.08,Z 331.95,A -85,B 0,C 180,E1 -21554.241,E2 -21554.241} C_VEL
LIN {X 0,Y 243.921,Z 316.892,A -85,B 0,C 180,E1 -21554.903,E2 -21554.903} C_VEL
LIN {X 0,Y 248.672,Z 242.907,A -85,B 0,C 180,E1 -21556.875,E2 -21556.875} C_VEL
LIN {X 0,Y 249.105,Z 233.497,A -85,B 0,C 180,E1 -21557.159,E2 -21557.159} C_VEL
LIN {X 0,Y 244.785,Z 224.182,A -85,B 0,C 180,E1 -21558.673,E2 -21558.673} C_VEL
LIN {X 0,Y 237.917,Z 212.394,A -85,B 0,C 180,E1 -21561.157,E2 -21561.157} C_VEL
LIN {X 0,Y 230.478,Z 200.811,A -85,B 0,C 180,E1 -21564.132,E2 -21564.132} C_VEL
LIN {X 0,Y 224.28,Z 191.956,A -85,B 0,C 180,E1 -21566.906,E2 -21566.906} C_VEL
LIN {X 0,Y 220.432,Z 186.929,A -85,B 0,C 180,E1 -21568.795,E2 -21568.795} C_VEL
LIN {X 0,Y 217.289,Z 182.801,A -85,B 0,C 180,E1 -21570.473,E2 -21570.473} C_VEL
LIN {X 0,Y 214.449,Z 179.359,A -85,B 0,C 180,E1 -21572.093,E2 -21572.093} C_VEL
LIN {X 0,Y 213.457,Z 177.968,A -85,B 0,C 180,E1 -21572.705,E2 -21572.705} C_VEL
LIN {X 0,Y 210.777,Z 175.191,A -85,B 0,C 180,E1 -21574.378,E2 -21574.378} C_VEL
LIN {X 0,Y 209.289,Z 172.759,A -85,B 0,C 180,E1 -21575.445,E2 -21575.445} C_VEL
LIN {X 0,Y 206.679,Z 170.699,A -85,B 0,C 180,E1 -21577.276,E2 -21577.276} C_VEL
LIN {X 0,Y 205.001,Z 167.851,A -85,B 0,C 180,E1 -21578.704,E2 -21578.704} C_VEL
LIN {X 0,Y 204.688,Z 167.154,A -85,B 0,C 180,E1 -21578.999,E2 -21578.999} C_VEL
LIN {X 0,Y 201.918,Z 165.551,A -85,B 0,C 180,E1 -21581.35,E2 -21581.35} C_VEL
LIN {X 0,Y 200.172,Z 162.942,A -85,B 0,C 180,E1 -21583.228,E2 -21583.228} C_VEL
LIN {X 0,Y 199.779,Z 161.226,A -85,B 0,C 180,E1 -21583.917,E2 -21583.917} C_VEL
LIN {X 0,Y 200.025,Z 161.182,A -85,B 0,C 180,E1 -21589.882,E2 -21589.882} C_VEL
LIN {X 0,Y 200.003,Z 161.19,A -85,B 0,C 180,E1 -21593.948,E2 -21593.948} C_VEL
LIN {X 0,Y 200.289,Z 161.161,A -85,B 0,C 180,E1 -21597.989,E2 -21597.989} C_VEL
LIN {X 0,Y 200.451,Z 161.126,A -85,B 0,C 180,E1 -21600,E2 -21600} C_VEL
LIN {X 0,Y 200.317,Z 161.156,A -85,B 0,C 180,E1 -21602.01,E2 -21602.01} C_VEL
LIN {X 0,Y 200.079,Z 161.18,A -85,B 0,C 180,E1 -21608.077,E2 -21608.077} C_VEL
LIN {X 0,Y 199.872,Z 161.211,A -85,B 0,C 180,E1 -21612.179,E2 -21612.179} C_VEL
LIN {X 0,Y 199.832,Z 161.276,A -85,B 0,C 180,E1 -21615.882,E2 -21615.882} C_VEL
LIN {X 0,Y 200.347,Z 163.23,A -85,B 0,C 180,E1 -21616.625,E2 -21616.625} C_VEL
LIN {X 0,Y 202.391,Z 165.908,A -85,B 0,C 180,E1 -21618.736,E2 -21618.736} C_VEL
LIN {X 0,Y 204.848,Z 167.33,A -85,B 0,C 180,E1 -21620.786,E2 -21620.786} C_VEL
LIN {X 0,Y 206.312,Z 170.207,A -85,B 0,C 180,E1 -21622.083,E2 -21622.083} C_VEL
LIN {X 0,Y 208.972,Z 172.592,A -85,B 0,C 180,E1 -21623.999,E2 -21623.999} C_VEL
LIN {X 0,Y 209.716,Z 173.249,A -85,B 0,C 180,E1 -21624.501,E2 -21624.501} C_VEL
LIN {X 0,Y 211.834,Z 176.461,A -85,B 0,C 180,E1 -21625.963,E2 -21625.963} C_VEL
LIN {X 0,Y 214.031,Z 178.63,A -85,B 0,C 180,E1 -21627.292,E2 -21627.292} C_VEL
LIN {X 0,Y 214.648,Z 179.705,A -85,B 0,C 180,E1 -21627.683,E2 -21627.683} C_VEL
LIN {X 0,Y 216.482,Z 183.34,A -85,B 0,C 180,E1 -21628.832,E2 -21628.832} C_VEL
LIN {X 0,Y 221.573,Z 198.299,A -85,B 0,C 180,E1 -21632.027,E2 -21632.027} C_VEL
LIN {X 0,Y 223.654,Z 202.096,A -85,B 0,C 180,E1 -21633.082,E2 -21633.082} C_VEL
LIN {X 0,Y 229.713,Z 212.753,A -85,B 0,C 180,E1 -21635.879,E2 -21635.879} C_VEL
LIN {X 0,Y 235.869,Z 224.839,A -85,B 0,C 180,E1 -21638.466,E2 -21638.466} C_VEL
LIN {X 0,Y 240.639,Z 235.314,A -85,B 0,C 180,E1 -21640.339,E2 -21640.339} C_VEL
LIN {X 0,Y 243.921,Z 243.303,A -85,B 0,C 180,E1 -21641.581,E2 -21641.581} C_VEL
LIN {X 0,Y 238.538,Z 325.61,A -85,B 0,C 180,E1 -21643.793,E2 -21643.793} C_VEL
LIN {X 0,Y 236.395,Z 341.749,A -85,B 0,C 180,E1 -21644.478,E2 -21644.478} C_VEL
LIN {X 0,Y 233.504,Z 356.996,A -85,B 0,C 180,E1 -21645.439,E2 -21645.439} C_VEL
LIN {X 0,Y 230.106,Z 370.73,A -85,B 0,C 180,E1 -21646.59,E2 -21646.59} C_VEL
LIN {X 0,Y 226.038,Z 384.816,A -85,B 0,C 180,E1 -21648.17,E2 -21648.17} C_VEL
LIN {X 0,Y 221.587,Z 397.9,A -85,B 0,C 180,E1 -21650.039,E2 -21650.039} C_VEL
LIN {X 0,Y 216.715,Z 410.316,A -85,B 0,C 180,E1 -21652.257,E2 -21652.257} C_VEL
LIN {X 0,Y 211.487,Z 422.495,A -85,B 0,C 180,E1 -21655.023,E2 -21655.023} C_VEL
LIN {X 0,Y 206.668,Z 433.07,A -85,B 0,C 180,E1 -21658.078,E2 -21658.078} C_VEL
LIN {X 0,Y 202.304,Z 442.377,A -85,B 0,C 180,E1 -21661.466,E2 -21661.466} C_VEL
LIN {X 0,Y 198.508,Z 449.877,A -85,B 0,C 180,E1 -21664.859,E2 -21664.859} C_VEL
LIN {X 0,Y 195.164,Z 456.882,A -85,B 0,C 180,E1 -21668.893,E2 -21668.893} C_VEL
LIN {X 0,Y 192.702,Z 462.397,A -85,B 0,C 180,E1 -21673.036,E2 -21673.036} C_VEL
LIN {X 0,Y 191.066,Z 466.572,A -85,B 0,C 180,E1 -21677.25,E2 -21677.25} C_VEL
LIN {X 0,Y 190.285,Z 469.508,A -85,B 0,C 180,E1 -21681.504,E2 -21681.504} C_VEL
LIN {X 0,Y 190.081,Z 471.263,A -85,B 0,C 180,E1 -21685.759,E2 -21685.759} C_VEL
LIN {X 0,Y 190.263,Z 471.867,A -85,B 0,C 180,E1 -21690,E2 -21690} C_VEL
LIN {X 0,Y 190.081,Z 471.247,A -85,B 0,C 180,E1 -21694.241,E2 -21694.241} C_VEL
LIN {X 0,Y 190.285,Z 469.472,A -85,B 0,C 180,E1 -21698.496,E2 -21698.496} C_VEL
LIN {X 0,Y 191.062,Z 466.52,A -85,B 0,C 180,E1 -21702.75,E2 -21702.75} C_VEL
LIN {X 0,Y 192.659,Z 462.33,A -85,B 0,C 180,E1 -21706.968,E2 -21706.968} C_VEL
LIN {X 0,Y 195.092,Z 456.789,A -85,B 0,C 180,E1 -21711.115,E2 -21711.115} C_VEL
LIN {X 0,Y 198.484,Z 449.754,A -85,B 0,C 180,E1 -21715.144,E2 -21715.144} C_VEL
LIN {X 0,Y 202.265,Z 442.24,A -85,B 0,C 180,E1 -21718.54,E2 -21718.54} C_VEL
LIN {X 0,Y 206.361,Z 433.383,A -85,B 0,C 180,E1 -21721.776,E2 -21721.776} C_VEL
LIN {X 0,Y 210.703,Z 423.938,A -85,B 0,C 180,E1 -21724.544,E2 -21724.544} C_VEL
LIN {X 0,Y 215.41,Z 413.058,A -85,B 0,C 180,E1 -21727.127,E2 -21727.127} C_VEL
LIN {X 0,Y 220.227,Z 401.19,A -85,B 0,C 180,E1 -21729.365,E2 -21729.365} C_VEL
LIN {X 0,Y 224.754,Z 388.352,A -85,B 0,C 180,E1 -21731.314,E2 -21731.314} C_VEL
LIN {X 0,Y 228.612,Z 375.629,A -85,B 0,C 180,E1 -21732.857,E2 -21732.857} C_VEL
LIN {X 0,Y 232.411,Z 360.976,A -85,B 0,C 180,E1 -21734.219,E2 -21734.219} C_VEL
LIN {X 0,Y 235.448,Z 346.365,A -85,B 0,C 180,E1 -21735.224,E2 -21735.224} C_VEL
LIN {X 0,Y 237.72,Z 331.404,A -85,B 0,C 180,E1 -21735.954,E2 -21735.954} C_VEL
LIN {X 0,Y 239.191,Z 314.546,A -85,B 0,C 180,E1 -21736.5,E2 -21736.5} C_VEL
LIN {X 0,Y 243.766,Z 243.06,A -85,B 0,C 180,E1 -21738.394,E2 -21738.394} C_VEL
LIN {X 0,Y 238.45,Z 230.554,A -85,B 0,C 180,E1 -21740.415,E2 -21740.415} C_VEL
LIN {X 0,Y 232.528,Z 218.253,A -85,B 0,C 180,E1 -21742.808,E2 -21742.808} C_VEL
LIN {X 0,Y 226.631,Z 207.261,A -85,B 0,C 180,E1 -21745.396,E2 -21745.396} C_VEL
LIN {X 0,Y 221.344,Z 198.247,A -85,B 0,C 180,E1 -21747.948,E2 -21747.948} C_VEL
LIN {X 0,Y 217.816,Z 192.912,A -85,B 0,C 180,E1 -21749.788,E2 -21749.788} C_VEL
LIN {X 0,Y 214.87,Z 188.924,A -85,B 0,C 180,E1 -21751.422,E2 -21751.422} C_VEL
LIN {X 0,Y 211.952,Z 185.154,A -85,B 0,C 180,E1 -21753.166,E2 -21753.166} C_VEL
LIN {X 0,Y 208.339,Z 180.86,A -85,B 0,C 180,E1 -21755.526,E2 -21755.526} C_VEL
LIN {X 0,Y 207.286,Z 179.272,A -85,B 0,C 180,E1 -21756.299,E2 -21756.299} C_VEL
LIN {X 0,Y 204.773,Z 176.927,A -85,B 0,C 180,E1 -21758.151,E2 -21758.151} C_VEL
LIN {X 0,Y 202.968,Z 173.901,A -85,B 0,C 180,E1 -21759.741,E2 -21759.741} C_VEL
LIN {X 0,Y 200.335,Z 172.074,A -85,B 0,C 180,E1 -21762.069,E2 -21762.069} C_VEL
LIN {X 0,Y 198.553,Z 169.14,A -85,B 0,C 180,E1 -21764.079,E2 -21764.079} C_VEL
LIN {X 0,Y 198.192,Z 168.124,A -85,B 0,C 180,E1 -21764.577,E2 -21764.577} C_VEL
LIN {X 0,Y 195.24,Z 166.567,A -85,B 0,C 180,E1 -21768.318,E2 -21768.318} C_VEL
LIN {X 0,Y 193.331,Z 163.463,A -85,B 0,C 180,E1 -21772.165,E2 -21772.165} C_VEL
LIN {X 0,Y 192.968,Z 162.072,A -85,B 0,C 180,E1 -21773.465,E2 -21773.465} C_VEL
LIN {X 0,Y 193.258,Z 162.038,A -85,B 0,C 180,E1 -21777.916,E2 -21777.916} C_VEL
LIN {X 0,Y 193.417,Z 162.004,A -85,B 0,C 180,E1 -21780,E2 -21780} C_VEL
LIN {X 0,Y 192.94,Z 162.064,A -85,B 0,C 180,E1 -21784.178,E2 -21784.178} C_VEL
LIN {X 0,Y 193.001,Z 162.244,A -85,B 0,C 180,E1 -21787.191,E2 -21787.191} C_VEL
LIN {X 0,Y 194.027,Z 164.995,A -85,B 0,C 180,E1 -21789.95,E2 -21789.95} C_VEL
LIN {X 0,Y 195.985,Z 167.198,A -85,B 0,C 180,E1 -21793.215,E2 -21793.215} C_VEL
LIN {X 0,Y 198.242,Z 168.384,A -85,B 0,C 180,E1 -21795.947,E2 -21795.947} C_VEL
LIN {X 0,Y 199.72,Z 171.397,A -85,B 0,C 180,E1 -21797.745,E2 -21797.745} C_VEL
LIN {X 0,Y 202.202,Z 173.57,A -85,B 0,C 180,E1 -21800.074,E2 -21800.074} C_VEL
LIN {X 0,Y 203.11,Z 174.121,A -85,B 0,C 180,E1 -21800.826,E2 -21800.826} C_VEL
LIN {X 0,Y 205.067,Z 177.411,A -85,B 0,C 180,E1 -21802.534,E2 -21802.534} C_VEL
LIN {X 0,Y 207.686,Z 179.714,A -85,B 0,C 180,E1 -21804.424,E2 -21804.424} C_VEL
LIN {X 0,Y 210.001,Z 183.127,A -85,B 0,C 180,E1 -21806.056,E2 -21806.056} C_VEL
LIN {X 0,Y 211.843,Z 185.039,A -85,B 0,C 180,E1 -21807.207,E2 -21807.207} C_VEL
LIN {X 0,Y 214.81,Z 188.932,A -85,B 0,C 180,E1 -21808.988,E2 -21808.988} C_VEL
LIN {X 0,Y 219.503,Z 195.145,A -85,B 0,C 180,E1 -21811.531,E2 -21811.531} C_VEL
LIN {X 0,Y 222.797,Z 199.799,A -85,B 0,C 180,E1 -21813.168,E2 -21813.168} C_VEL
LIN {X 0,Y 227.916,Z 207.319,A -85,B 0,C 180,E1 -21815.508,E2 -21815.508} C_VEL
LIN {X 0,Y 234.204,Z 217.299,A -85,B 0,C 180,E1 -21818.117,E2 -21818.117} C_VEL
LIN {X 0,Y 241.443,Z 230.05,A -85,B 0,C 180,E1 -21820.846,E2 -21820.846} C_VEL
LIN {X 0,Y 244.103,Z 236.043,A -85,B 0,C 180,E1 -21821.83,E2 -21821.83} C_VEL
LIN {X 0,Y 238.968,Z 315.516,A -85,B 0,C 180,E1 -21823.977,E2 -21823.977} C_VEL
LIN {X 0,Y 236.994,Z 331.146,A -85,B 0,C 180,E1 -21824.625,E2 -21824.625} C_VEL
LIN {X 0,Y 234.57,Z 345.45,A -85,B 0,C 180,E1 -21825.545,E2 -21825.545} C_VEL
LIN {X 0,Y 231.361,Z 360.032,A -85,B 0,C 180,E1 -21826.806,E2 -21826.806} C_VEL
LIN {X 0,Y 227.573,Z 374.089,A -85,B 0,C 180,E1 -21828.396,E2 -21828.396} C_VEL
LIN {X 0,Y 223.492,Z 386.555,A -85,B 0,C 180,E1 -21830.154,E2 -21830.154} C_VEL
LIN {X 0,Y 219.14,Z 398.123,A -85,B 0,C 180,E1 -21832.167,E2 -21832.167} C_VEL
LIN {X 0,Y 214.663,Z 408.867,A -85,B 0,C 180,E1 -21834.47,E2 -21834.47} C_VEL
LIN {X 0,Y 210.624,Z 418.142,A -85,B 0,C 180,E1 -21836.914,E2 -21836.914} C_VEL
LIN {X 0,Y 206.285,Z 427.225,A -85,B 0,C 180,E1 -21839.833,E2 -21839.833} C_VEL
LIN {X 0,Y 202.197,Z 435.476,A -85,B 0,C 180,E1 -21843.137,E2 -21843.137} C_VEL
LIN {X 0,Y 198.161,Z 443.225,A -85,B 0,C 180,E1 -21847.038,E2 -21847.038} C_VEL
LIN {X 0,Y 195.196,Z 449.38,A -85,B 0,C 180,E1 -21851.092,E2 -21851.092} C_VEL
LIN {X 0,Y 192.889,Z 454.13,A -85,B 0,C 180,E1 -21855.224,E2 -21855.224} C_VEL
LIN {X 0,Y 191.455,Z 457.601,A -85,B 0,C 180,E1 -21859.424,E2 -21859.424} C_VEL
LIN {X 0,Y 190.598,Z 459.893,A -85,B 0,C 180,E1 -21863.649,E2 -21863.649} C_VEL
LIN {X 0,Y 190.279,Z 461.057,A -85,B 0,C 180,E1 -21867.883,E2 -21867.883} C_VEL
LIN {X 0,Y 190.301,Z 461.211,A -85,B 0,C 180,E1 -21870,E2 -21870} C_VEL
LIN {X 0,Y 190.444,Z 460.499,A -85,B 0,C 180,E1 -21874.869,E2 -21874.869} C_VEL
LIN {X 0,Y 190.929,Z 458.975,A -85,B 0,C 180,E1 -21878.467,E2 -21878.467} C_VEL
LIN {X 0,Y 192.019,Z 456.147,A -85,B 0,C 180,E1 -21882.686,E2 -21882.686} C_VEL
